LIN {X 0,Y 194.832,Z 950.293,A -85,B 0,C 180,E1 7671.992,E2 7671.992} C_VEL
LIN {X 0,Y 183.693,Z 961.41,A -85,B 0,C 180,E1 7666.758,E2 7666.758} C_VEL
LIN {X 0,Y 173.578,Z 971.355,A -85,B 0,C 180,E1 7660.613,E2 7660.613} C_VEL
LIN {X 0,Y 165.361,Z 979.416,A -85,B 0,C 180,E1 7653.893,E2 7653.893} C_VEL
LIN {X 0,Y 158.738,Z 986.366,A -85,B 0,C 180,E1 7646.018,E2 7646.018} C_VEL
LIN {X 0,Y 154.956,Z 990.985,A -85,B 0,C 180,E1 7638.756,E2 7638.756} C_VEL
LIN {X 0,Y 152.752,Z 994.605,A -85,B 0,C 180,E1 7630.489,E2 7630.489} C_VEL
LIN {X 0,Y 152.139,Z 996.368,A -85,B 0,C 180,E1 7623.866,E2 7623.866} C_VEL
LIN {X 0,Y 152.069,Z 997.179,A -85,B 0,C 180,E1 7618.016,E2 7618.016} C_VEL
LIN {X 0,Y 152.181,Z 997.294,A -85,B 0,C 180,E1 7612.04,E2 7612.04} C_VEL
LIN {X 0,Y 152.864,Z 996.613,A -85,B 0,C 180,E1 7605.477,E2 7605.477} C_VEL
LIN {X 0,Y 155.417,Z 994.355,A -85,B 0,C 180,E1 7596.75,E2 7596.75} C_VEL
LIN {X 0,Y 159.971,Z 990.88,A -85,B 0,C 180,E1 7588.935,E2 7588.935} C_VEL
LIN {X 0,Y 168.381,Z 984.987,A -85,B 0,C 180,E1 7580.226,E2 7580.226} C_VEL
LIN {X 0,Y 178.983,Z 977.818,A -85,B 0,C 180,E1 7572.913,E2 7572.913} C_VEL
LIN {X 0,Y 191.582,Z 968.945,A -85,B 0,C 180,E1 7566.594,E2 7566.594} C_VEL
LIN {X 0,Y 207.009,Z 957.677,A -85,B 0,C 180,E1 7560.794,E2 7560.794} C_VEL
LIN {X 0,Y 222.449,Z 945.698,A -85,B 0,C 180,E1 7556.307,E2 7556.307} C_VEL
LIN {X 0,Y 238.515,Z 932.053,A -85,B 0,C 180,E1 7552.534,E2 7552.534} C_VEL
LIN {X 0,Y 255.431,Z 916.454,A -85,B 0,C 180,E1 7549.29,E2 7549.29} C_VEL
LIN {X 0,Y 271.677,Z 899.924,A -85,B 0,C 180,E1 7546.703,E2 7546.703} C_VEL
LIN {X 0,Y 286.835,Z 882.673,A -85,B 0,C 180,E1 7544.638,E2 7544.638} C_VEL
LIN {X 0,Y 271.407,Z 900.775,A -85,B 0,C 180,E1 7542.66,E2 7542.66} C_VEL
LIN {X 0,Y 266.25,Z 906.214,A -85,B 0,C 180,E1 7542.181,E2 7542.181} C_VEL
LIN {X 0,Y 251.976,Z 920.113,A -85,B 0,C 180,E1 7541.531,E2 7541.531} C_VEL
LIN {X 0,Y 246.66,Z 924.954,A -85,B 0,C 180,E1 7540.925,E2 7540.925} C_VEL
LIN {X 0,Y 229.187,Z 940.666,A -85,B 0,C 180,E1 7537.662,E2 7537.662} C_VEL
LIN {X 0,Y 212.755,Z 954.165,A -85,B 0,C 180,E1 7533.859,E2 7533.859} C_VEL
LIN {X 0,Y 195.426,Z 967.538,A -85,B 0,C 180,E1 7528.708,E2 7528.708} C_VEL
LIN {X 0,Y 181.211,Z 978.023,A -85,B 0,C 180,E1 7523.147,E2 7523.147} C_VEL
LIN {X 0,Y 168.432,Z 987.146,A -85,B 0,C 180,E1 7516.415,E2 7516.415} C_VEL
LIN {X 0,Y 158.156,Z 994.699,A -85,B 0,C 180,E1 7508.757,E2 7508.757} C_VEL
LIN {X 0,Y 150.669,Z 1000.453,A -85,B 0,C 180,E1 7500.298,E2 7500.298} C_VEL
LIN {X 0,Y 146.133,Z 1004.752,A -85,B 0,C 180,E1 7491.272,E2 7491.272} C_VEL
LIN {X 0,Y 144.3,Z 1007.131,A -85,B 0,C 180,E1 7482.821,E2 7482.821} C_VEL
LIN {X 0,Y 144.029,Z 1008.079,A -85,B 0,C 180,E1 7476.387,E2 7476.387} C_VEL
LIN {X 0,Y 144.076,Z 1008.216,A -85,B 0,C 180,E1 7470.408,E2 7470.408} C_VEL
LIN {X 0,Y 144.045,Z 1007.654,A -85,B 0,C 180,E1 7464.833,E2 7464.833} C_VEL
LIN {X 0,Y 144.179,Z 1006.3,A -85,B 0,C 180,E1 7458.814,E2 7458.814} C_VEL
LIN {X 0,Y 145.28,Z 1003.668,A -85,B 0,C 180,E1 7451.555,E2 7451.555} C_VEL
LIN {X 0,Y 148.668,Z 998.874,A -85,B 0,C 180,E1 7442.797,E2 7442.797} C_VEL
LIN {X 0,Y 153.972,Z 992.973,A -85,B 0,C 180,E1 7435.162,E2 7435.162} C_VEL
LIN {X 0,Y 162.295,Z 984.672,A -85,B 0,C 180,E1 7427.352,E2 7427.352} C_VEL
LIN {X 0,Y 172.502,Z 974.948,A -85,B 0,C 180,E1 7420.613,E2 7420.613} C_VEL
LIN {X 0,Y 184.018,Z 963.646,A -85,B 0,C 180,E1 7414.887,E2 7414.887} C_VEL
LIN {X 0,Y 196.383,Z 951.126,A -85,B 0,C 180,E1 7410.075,E2 7410.075} C_VEL
LIN {X 0,Y 208.775,Z 937.625,A -85,B 0,C 180,E1 7406.141,E2 7406.141} C_VEL
LIN {X 0,Y 223.027,Z 920.827,A -85,B 0,C 180,E1 7402.399,E2 7402.399} C_VEL
LIN {X 0,Y 235.885,Z 904.265,A -85,B 0,C 180,E1 7399.563,E2 7399.563} C_VEL
LIN {X 0,Y 248.354,Z 886.236,A -85,B 0,C 180,E1 7397.176,E2 7397.176} C_VEL
LIN {X 0,Y 260.04,Z 867.469,A -85,B 0,C 180,E1 7395.211,E2 7395.211} C_VEL
LIN {X 0,Y 270.544,Z 848.252,A -85,B 0,C 180,E1 7393.628,E2 7393.628} C_VEL
LIN {X 0,Y 280.799,Z 826.787,A -85,B 0,C 180,E1 7392.231,E2 7392.231} C_VEL
LIN {X 0,Y 289.504,Z 805.535,A -85,B 0,C 180,E1 7391.151,E2 7391.151} C_VEL
LIN {X 0,Y 297.135,Z 782.995,A -85,B 0,C 180,E1 7390.273,E2 7390.273} C_VEL
LIN {X 0,Y 303.574,Z 759.689,A -85,B 0,C 180,E1 7389.596,E2 7389.596} C_VEL
LIN {X 0,Y 308.243,Z 736.843,A -85,B 0,C 180,E1 7389.078,E2 7389.078} C_VEL
LIN {X 0,Y 312.449,Z 705.289,A -85,B 0,C 180,E1 7388.469,E2 7388.469} C_VEL
LIN {X 0,Y 324.295,Z 602.682,A -85,B 0,C 180,E1 7386.606,E2 7386.606} C_VEL
LIN {X 0,Y 320.232,Z 595.927,A -85,B 0,C 180,E1 7383.132,E2 7383.132} C_VEL
LIN {X 0,Y 317.949,Z 592.19,A -85,B 0,C 180,E1 7380.805,E2 7380.805} C_VEL
LIN {X 0,Y 315.597,Z 588.414,A -85,B 0,C 180,E1 7378.002,E2 7378.002} C_VEL
LIN {X 0,Y 312.963,Z 584.083,A -85,B 0,C 180,E1 7373.948,E2 7373.948} C_VEL
LIN {X 0,Y 310.602,Z 579.992,A -85,B 0,C 180,E1 7367.23,E2 7367.23} C_VEL
LIN {X 0,Y 310.395,Z 579.187,A -85,B 0,C 180,E1 7365.447,E2 7365.447} C_VEL
LIN {X 0,Y 310.527,Z 579.358,A -85,B 0,C 180,E1 7360.826,E2 7360.826} C_VEL
LIN {X 0,Y 312.556,Z 583.694,A -85,B 0,C 180,E1 7354.007,E2 7354.007} C_VEL
LIN {X 0,Y 313.453,Z 584.799,A -85,B 0,C 180,E1 7352.449,E2 7352.449} C_VEL
LIN {X 0,Y 316.52,Z 589.805,A -85,B 0,C 180,E1 7348.054,E2 7348.054} C_VEL
LIN {X 0,Y 319.481,Z 594.635,A -85,B 0,C 180,E1 7344.84,E2 7344.84} C_VEL
LIN {X 0,Y 323.414,Z 601.079,A -85,B 0,C 180,E1 7341.354,E2 7341.354} C_VEL
LIN {X 0,Y 323.931,Z 602.297,A -85,B 0,C 180,E1 7340.903,E2 7340.903} C_VEL
LIN {X 0,Y 309.802,Z 722.184,A -85,B 0,C 180,E1 7338.744,E2 7338.744} C_VEL
LIN {X 0,Y 305.322,Z 746.033,A -85,B 0,C 180,E1 7338.204,E2 7338.204} C_VEL
LIN {X 0,Y 299.821,Z 768.228,A -85,B 0,C 180,E1 7337.538,E2 7337.538} C_VEL
LIN {X 0,Y 292.969,Z 789.815,A -85,B 0,C 180,E1 7336.686,E2 7336.686} C_VEL
LIN {X 0,Y 284.325,Z 812.53,A -85,B 0,C 180,E1 7335.541,E2 7335.541} C_VEL
LIN {X 0,Y 275.54,Z 832.057,A -85,B 0,C 180,E1 7334.299,E2 7334.299} C_VEL
LIN {X 0,Y 264.822,Z 852.675,A -85,B 0,C 180,E1 7332.656,E2 7332.656} C_VEL
LIN {X 0,Y 253.514,Z 871.813,A -85,B 0,C 180,E1 7330.738,E2 7330.738} C_VEL
LIN {X 0,Y 241.283,Z 889.944,A -85,B 0,C 180,E1 7328.423,E2 7328.423} C_VEL
LIN {X 0,Y 228.308,Z 907.306,A -85,B 0,C 180,E1 7325.614,E2 7325.614} C_VEL
LIN {X 0,Y 215.842,Z 922.349,A -85,B 0,C 180,E1 7322.494,E2 7322.494} C_VEL
LIN {X 0,Y 202.641,Z 936.953,A -85,B 0,C 180,E1 7318.585,E2 7318.585} C_VEL
LIN {X 0,Y 190.981,Z 948.948,A -85,B 0,C 180,E1 7314.421,E2 7314.421} C_VEL
LIN {X 0,Y 178.697,Z 960.792,A -85,B 0,C 180,E1 7308.982,E2 7308.982} C_VEL
LIN {X 0,Y 167.816,Z 971.009,A -85,B 0,C 180,E1 7302.726,E2 7302.726} C_VEL
LIN {X 0,Y 158.765,Z 979.33,A -85,B 0,C 180,E1 7295.698,E2 7295.698} C_VEL
LIN {X 0,Y 151.411,Z 986.537,A -85,B 0,C 180,E1 7287.341,E2 7287.341} C_VEL
LIN {X 0,Y 147.3,Z 991.142,A -85,B 0,C 180,E1 7279.823,E2 7279.823} C_VEL
LIN {X 0,Y 144.836,Z 994.849,A -85,B 0,C 180,E1 7271.047,E2 7271.047} C_VEL
LIN {X 0,Y 144.152,Z 996.634,A -85,B 0,C 180,E1 7264.078,E2 7264.078} C_VEL
LIN {X 0,Y 144.072,Z 997.476,A -85,B 0,C 180,E1 7257.854,E2 7257.854} C_VEL
LIN {X 0,Y 144.21,Z 997.615,A -85,B 0,C 180,E1 7251.581,E2 7251.581} C_VEL
LIN {X 0,Y 144.995,Z 996.975,A -85,B 0,C 180,E1 7244.7,E2 7244.7} C_VEL
LIN {X 0,Y 147.862,Z 994.811,A -85,B 0,C 180,E1 7235.561,E2 7235.561} C_VEL
LIN {X 0,Y 153.044,Z 991.301,A -85,B 0,C 180,E1 7227.216,E2 7227.216} C_VEL
LIN {X 0,Y 162.181,Z 985.516,A -85,B 0,C 180,E1 7218.277,E2 7218.277} C_VEL
LIN {X 0,Y 173.324,Z 978.573,A -85,B 0,C 180,E1 7210.975,E2 7210.975} C_VEL
LIN {X 0,Y 186.679,Z 969.849,A -85,B 0,C 180,E1 7204.609,E2 7204.609} C_VEL
LIN {X 0,Y 201.882,Z 959.492,A -85,B 0,C 180,E1 7199.15,E2 7199.15} C_VEL
LIN {X 0,Y 216.832,Z 948.494,A -85,B 0,C 180,E1 7194.941,E2 7194.941} C_VEL
LIN {X 0,Y 234.646,Z 934.325,A -85,B 0,C 180,E1 7190.93,E2 7190.93} C_VEL
LIN {X 0,Y 251.632,Z 919.547,A -85,B 0,C 180,E1 7187.836,E2 7187.836} C_VEL
LIN {X 0,Y 268.871,Z 902.747,A -85,B 0,C 180,E1 7185.224,E2 7185.224} C_VEL
LIN {X 0,Y 272.667,Z 898.907,A -85,B 0,C 180,E1 7184.682,E2 7184.682} C_VEL
LIN {X 0,Y 256.832,Z 915.179,A -85,B 0,C 180,E1 7182.528,E2 7182.528} C_VEL
LIN {X 0,Y 246.66,Z 924.954,A -85,B 0,C 180,E1 7180.925,E2 7180.925} C_VEL
LIN {X 0,Y 241.229,Z 929.896,A -85,B 0,C 180,E1 7180.269,E2 7180.269} C_VEL
LIN {X 0,Y 225.887,Z 942.079,A -85,B 0,C 180,E1 7179.184,E2 7179.184} C_VEL
LIN {X 0,Y 220.354,Z 946.366,A -85,B 0,C 180,E1 7178.369,E2 7178.369} C_VEL
LIN {X 0,Y 202.342,Z 960.072,A -85,B 0,C 180,E1 7174.084,E2 7174.084} C_VEL
LIN {X 0,Y 185.384,Z 972.199,A -85,B 0,C 180,E1 7168.818,E2 7168.818} C_VEL
LIN {X 0,Y 170.774,Z 981.996,A -85,B 0,C 180,E1 7162.786,E2 7162.786} C_VEL
LIN {X 0,Y 157.16,Z 991.006,A -85,B 0,C 180,E1 7154.937,E2 7154.937} C_VEL
LIN {X 0,Y 147.801,Z 997.325,A -85,B 0,C 180,E1 7147.03,E2 7147.03} C_VEL
LIN {X 0,Y 140.534,Z 1002.714,A -85,B 0,C 180,E1 7137.098,E2 7137.098} C_VEL
LIN {X 0,Y 137.2,Z 1005.822,A -85,B 0,C 180,E1 7128.273,E2 7128.273} C_VEL
LIN {X 0,Y 136.079,Z 1007.586,A -85,B 0,C 180,E1 7119.313,E2 7119.313} C_VEL
LIN {X 0,Y 136.056,Z 1007.968,A -85,B 0,C 180,E1 7112.538,E2 7112.538} C_VEL
LIN {X 0,Y 136.056,Z 1007.622,A -85,B 0,C 180,E1 7106.641,E2 7106.641} C_VEL
LIN {X 0,Y 136.145,Z 1006.248,A -85,B 0,C 180,E1 7099.432,E2 7099.432} C_VEL
LIN {X 0,Y 137.195,Z 1003.721,A -85,B 0,C 180,E1 7091.749,E2 7091.749} C_VEL
LIN {X 0,Y 140.484,Z 999.348,A -85,B 0,C 180,E1 7082.827,E2 7082.827} C_VEL
LIN {X 0,Y 146.158,Z 993.337,A -85,B 0,C 180,E1 7074.459,E2 7074.459} C_VEL
LIN {X 0,Y 154.826,Z 985.253,A -85,B 0,C 180,E1 7066.306,E2 7066.306} C_VEL
LIN {X 0,Y 164.335,Z 976.602,A -85,B 0,C 180,E1 7059.965,E2 7059.965} C_VEL
LIN {X 0,Y 177.145,Z 964.76,A -85,B 0,C 180,E1 7053.581,E2 7053.581} C_VEL
LIN {X 0,Y 190.24,Z 952.141,A -85,B 0,C 180,E1 7048.572,E2 7048.572} C_VEL
LIN {X 0,Y 203.298,Z 938.468,A -85,B 0,C 180,E1 7044.535,E2 7044.535} C_VEL
LIN {X 0,Y 216.778,Z 923.303,A -85,B 0,C 180,E1 7041.085,E2 7041.085} C_VEL
LIN {X 0,Y 229.876,Z 906.972,A -85,B 0,C 180,E1 7038.249,E2 7038.249} C_VEL
LIN {X 0,Y 243.433,Z 888.208,A -85,B 0,C 180,E1 7035.728,E2 7035.728} C_VEL
LIN {X 0,Y 255.742,Z 869.143,A -85,B 0,C 180,E1 7033.734,E2 7033.734} C_VEL
LIN {X 0,Y 267.046,Z 849.002,A -85,B 0,C 180,E1 7032.102,E2 7032.102} C_VEL
LIN {X 0,Y 277.766,Z 827.118,A -85,B 0,C 180,E1 7030.713,E2 7030.713} C_VEL
LIN {X 0,Y 286.504,Z 806.21,A -85,B 0,C 180,E1 7029.681,E2 7029.681} C_VEL
LIN {X 0,Y 294.402,Z 783.436,A -85,B 0,C 180,E1 7028.819,E2 7028.819} C_VEL
LIN {X 0,Y 300.942,Z 760.311,A -85,B 0,C 180,E1 7028.167,E2 7028.167} C_VEL
LIN {X 0,Y 305.784,Z 737.07,A -85,B 0,C 180,E1 7027.657,E2 7027.657} C_VEL
LIN {X 0,Y 310.085,Z 705.601,A -85,B 0,C 180,E1 7027.063,E2 7027.063} C_VEL
LIN {X 0,Y 321.529,Z 608.329,A -85,B 0,C 180,E1 7025.352,E2 7025.352} C_VEL
LIN {X 0,Y 317.312,Z 601.015,A -85,B 0,C 180,E1 7021.354,E2 7021.354} C_VEL
LIN {X 0,Y 314.291,Z 596.237,A -85,B 0,C 180,E1 7017.812,E2 7017.812} C_VEL
LIN {X 0,Y 311.709,Z 591.924,A -85,B 0,C 180,E1 7013.738,E2 7013.738} C_VEL
LIN {X 0,Y 309.455,Z 587.902,A -85,B 0,C 180,E1 7007.118,E2 7007.118} C_VEL
LIN {X 0,Y 309.262,Z 587.103,A -85,B 0,C 180,E1 7005.393,E2 7005.393} C_VEL
LIN {X 0,Y 309.401,Z 587.346,A -85,B 0,C 180,E1 7000.754,E2 7000.754} C_VEL
LIN {X 0,Y 311.174,Z 591.374,A -85,B 0,C 180,E1 6994.496,E2 6994.496} C_VEL
LIN {X 0,Y 312.197,Z 592.659,A -85,B 0,C 180,E1 6992.639,E2 6992.639} C_VEL
LIN {X 0,Y 315.136,Z 597.553,A -85,B 0,C 180,E1 6988.325,E2 6988.325} C_VEL
LIN {X 0,Y 318.002,Z 602.339,A -85,B 0,C 180,E1 6985.137,E2 6985.137} C_VEL
LIN {X 0,Y 321.19,Z 607.752,A -85,B 0,C 180,E1 6982.187,E2 6982.187} C_VEL
LIN {X 0,Y 307.433,Z 722.444,A -85,B 0,C 180,E1 6980.162,E2 6980.162} C_VEL
LIN {X 0,Y 302.898,Z 746.237,A -85,B 0,C 180,E1 6979.641,E2 6979.641} C_VEL
LIN {X 0,Y 297.363,Z 768.273,A -85,B 0,C 180,E1 6979.003,E2 6979.003} C_VEL
LIN {X 0,Y 290.411,Z 789.843,A -85,B 0,C 180,E1 6978.182,E2 6978.182} C_VEL
LIN {X 0,Y 281.81,Z 812.156,A -85,B 0,C 180,E1 6977.1,E2 6977.1} C_VEL
LIN {X 0,Y 272.857,Z 831.753,A -85,B 0,C 180,E1 6975.898,E2 6975.898} C_VEL
LIN {X 0,Y 261.699,Z 852.86,A -85,B 0,C 180,E1 6974.27,E2 6974.27} C_VEL
LIN {X 0,Y 249.952,Z 872.361,A -85,B 0,C 180,E1 6972.369,E2 6972.369} C_VEL
LIN {X 0,Y 237.434,Z 890.496,A -85,B 0,C 180,E1 6970.103,E2 6970.103} C_VEL
LIN {X 0,Y 224.118,Z 907.857,A -85,B 0,C 180,E1 6967.344,E2 6967.344} C_VEL
LIN {X 0,Y 211.285,Z 922.885,A -85,B 0,C 180,E1 6964.263,E2 6964.263} C_VEL
LIN {X 0,Y 197.639,Z 937.451,A -85,B 0,C 180,E1 6960.381,E2 6960.381} C_VEL
LIN {X 0,Y 184.89,Z 950.09,A -85,B 0,C 180,E1 6955.969,E2 6955.969} C_VEL
LIN {X 0,Y 172.619,Z 961.369,A -85,B 0,C 180,E1 6950.681,E2 6950.681} C_VEL
LIN {X 0,Y 161.281,Z 971.477,A -85,B 0,C 180,E1 6944.348,E2 6944.348} C_VEL
LIN {X 0,Y 151.792,Z 979.707,A -85,B 0,C 180,E1 6937.179,E2 6937.179} C_VEL
LIN {X 0,Y 143.882,Z 986.946,A -85,B 0,C 180,E1 6928.397,E2 6928.397} C_VEL
LIN {X 0,Y 139.484,Z 991.535,A -85,B 0,C 180,E1 6920.5,E2 6920.5} C_VEL
LIN {X 0,Y 136.856,Z 995.203,A -85,B 0,C 180,E1 6911.238,E2 6911.238} C_VEL
LIN {X 0,Y 136.147,Z 996.973,A -85,B 0,C 180,E1 6903.844,E2 6903.844} C_VEL
LIN {X 0,Y 136.075,Z 997.777,A -85,B 0,C 180,E1 6897.55,E2 6897.55} C_VEL
LIN {X 0,Y 136.243,Z 997.939,A -85,B 0,C 180,E1 6891.072,E2 6891.072} C_VEL
LIN {X 0,Y 137.162,Z 997.335,A -85,B 0,C 180,E1 6883.794,E2 6883.794} C_VEL
LIN {X 0,Y 140.373,Z 995.277,A -85,B 0,C 180,E1 6874.245,E2 6874.245} C_VEL
LIN {X 0,Y 146.175,Z 991.795,A -85,B 0,C 180,E1 6865.438,E2 6865.438} C_VEL
LIN {X 0,Y 156.187,Z 986.085,A -85,B 0,C 180,E1 6856.181,E2 6856.181} C_VEL
LIN {X 0,Y 168.818,Z 978.845,A -85,B 0,C 180,E1 6848.424,E2 6848.424} C_VEL
LIN {X 0,Y 183.116,Z 970.124,A -85,B 0,C 180,E1 6842.097,E2 6842.097} C_VEL
LIN {X 0,Y 199.318,Z 959.7,A -85,B 0,C 180,E1 6836.715,E2 6836.715} C_VEL
LIN {X 0,Y 215.447,Z 948.401,A -85,B 0,C 180,E1 6832.535,E2 6832.535} C_VEL
LIN {X 0,Y 233.421,Z 934.669,A -85,B 0,C 180,E1 6828.812,E2 6828.812} C_VEL
LIN {X 0,Y 250.67,Z 920.224,A -85,B 0,C 180,E1 6825.919,E2 6825.919} C_VEL
LIN {X 0,Y 258.508,Z 913.046,A -85,B 0,C 180,E1 6824.752,E2 6824.752} C_VEL
LIN {X 0,Y 241.477,Z 928.765,A -85,B 0,C 180,E1 6822.252,E2 6822.252} C_VEL
LIN {X 0,Y 223.758,Z 943.608,A -85,B 0,C 180,E1 6819.066,E2 6819.066} C_VEL
LIN {X 0,Y 220.354,Z 946.366,A -85,B 0,C 180,E1 6818.369,E2 6818.369} C_VEL
LIN {X 0,Y 214.771,Z 950.617,A -85,B 0,C 180,E1 6817.487,E2 6817.487} C_VEL
LIN {X 0,Y 198.781,Z 961.182,A -85,B 0,C 180,E1 6815.791,E2 6815.791} C_VEL
LIN {X 0,Y 193.104,Z 964.791,A -85,B 0,C 180,E1 6814.666,E2 6814.666} C_VEL
LIN {X 0,Y 176.188,Z 975.809,A -85,B 0,C 180,E1 6809.288,E2 6809.288} C_VEL
LIN {X 0,Y 159.726,Z 986.02,A -85,B 0,C 180,E1 6802.081,E2 6802.081} C_VEL
LIN {X 0,Y 146.511,Z 994.111,A -85,B 0,C 180,E1 6793.666,E2 6793.666} C_VEL
LIN {X 0,Y 136.907,Z 1000.051,A -85,B 0,C 180,E1 6784.23,E2 6784.23} C_VEL
LIN {X 0,Y 130.704,Z 1004.496,A -85,B 0,C 180,E1 6773.371,E2 6773.371} C_VEL
LIN {X 0,Y 128.478,Z 1006.637,A -85,B 0,C 180,E1 6764.432,E2 6764.432} C_VEL
LIN {X 0,Y 128.037,Z 1007.576,A -85,B 0,C 180,E1 6756.288,E2 6756.288} C_VEL
LIN {X 0,Y 128.09,Z 1007.539,A -85,B 0,C 180,E1 6749.565,E2 6749.565} C_VEL
LIN {X 0,Y 128.05,Z 1006.691,A -85,B 0,C 180,E1 6742.582,E2 6742.582} C_VEL
LIN {X 0,Y 128.77,Z 1004.438,A -85,B 0,C 180,E1 6733.781,E2 6733.781} C_VEL
LIN {X 0,Y 131.207,Z 1000.907,A -85,B 0,C 180,E1 6725.234,E2 6725.234} C_VEL
LIN {X 0,Y 136.395,Z 995.606,A -85,B 0,C 180,E1 6716.157,E2 6716.157} C_VEL
LIN {X 0,Y 144.237,Z 988.47,A -85,B 0,C 180,E1 6707.763,E2 6707.763} C_VEL
LIN {X 0,Y 154.54,Z 979.684,A -85,B 0,C 180,E1 6700.248,E2 6700.248} C_VEL
LIN {X 0,Y 165.702,Z 969.975,A -85,B 0,C 180,E1 6694.261,E2 6694.261} C_VEL
LIN {X 0,Y 179.743,Z 957.256,A -85,B 0,C 180,E1 6688.511,E2 6688.511} C_VEL
LIN {X 0,Y 192.967,Z 944.44,A -85,B 0,C 180,E1 6684.248,E2 6684.248} C_VEL
LIN {X 0,Y 207.087,Z 929.495,A -85,B 0,C 180,E1 6680.527,E2 6680.527} C_VEL
LIN {X 0,Y 220.687,Z 913.83,A -85,B 0,C 180,E1 6677.532,E2 6677.532} C_VEL
LIN {X 0,Y 233.937,Z 896.685,A -85,B 0,C 180,E1 6675.03,E2 6675.03} C_VEL
LIN {X 0,Y 247.299,Z 877.408,A -85,B 0,C 180,E1 6672.848,E2 6672.848} C_VEL
LIN {X 0,Y 258.846,Z 858.522,A -85,B 0,C 180,E1 6671.186,E2 6671.186} C_VEL
LIN {X 0,Y 269.837,Z 837.889,A -85,B 0,C 180,E1 6669.766,E2 6669.766} C_VEL
LIN {X 0,Y 279.521,Z 817.029,A -85,B 0,C 180,E1 6668.64,E2 6668.64} C_VEL
LIN {X 0,Y 288.038,Z 794.958,A -85,B 0,C 180,E1 6667.727,E2 6667.727} C_VEL
LIN {X 0,Y 295.615,Z 771.189,A -85,B 0,C 180,E1 6666.985,E2 6666.985} C_VEL
LIN {X 0,Y 301.259,Z 748.585,A -85,B 0,C 180,E1 6666.451,E2 6666.451} C_VEL
LIN {X 0,Y 305.459,Z 724.638,A -85,B 0,C 180,E1 6665.976,E2 6665.976} C_VEL
LIN {X 0,Y 318.866,Z 614.103,A -85,B 0,C 180,E1 6664.045,E2 6664.045} C_VEL
LIN {X 0,Y 315.202,Z 607.785,A -85,B 0,C 180,E1 6660.363,E2 6660.363} C_VEL
LIN {X 0,Y 312.845,Z 603.886,A -85,B 0,C 180,E1 6657.435,E2 6657.435} C_VEL
LIN {X 0,Y 310.459,Z 599.764,A -85,B 0,C 180,E1 6653.527,E2 6653.527} C_VEL
LIN {X 0,Y 308.303,Z 595.714,A -85,B 0,C 180,E1 6646.878,E2 6646.878} C_VEL
LIN {X 0,Y 308.101,Z 594.982,A -85,B 0,C 180,E1 6644.952,E2 6644.952} C_VEL
LIN {X 0,Y 308.26,Z 595.245,A -85,B 0,C 180,E1 6640.876,E2 6640.876} C_VEL
LIN {X 0,Y 310.088,Z 599.376,A -85,B 0,C 180,E1 6634.4,E2 6634.4} C_VEL
LIN {X 0,Y 310.937,Z 600.517,A -85,B 0,C 180,E1 6632.83,E2 6632.83} C_VEL
LIN {X 0,Y 313.751,Z 605.286,A -85,B 0,C 180,E1 6628.608,E2 6628.608} C_VEL
LIN {X 0,Y 316.502,Z 609.991,A -85,B 0,C 180,E1 6625.465,E2 6625.465} C_VEL
LIN {X 0,Y 318.537,Z 613.657,A -85,B 0,C 180,E1 6623.475,E2 6623.475} C_VEL
LIN {X 0,Y 305.142,Z 722.86,A -85,B 0,C 180,E1 6621.594,E2 6621.594} C_VEL
LIN {X 0,Y 300.517,Z 746.67,A -85,B 0,C 180,E1 6621.089,E2 6621.089} C_VEL
LIN {X 0,Y 294.648,Z 769.471,A -85,B 0,C 180,E1 6620.447,E2 6620.447} C_VEL
LIN {X 0,Y 287.809,Z 790.341,A -85,B 0,C 180,E1 6619.679,E2 6619.679} C_VEL
LIN {X 0,Y 278.977,Z 812.85,A -85,B 0,C 180,E1 6618.622,E2 6618.622} C_VEL
LIN {X 0,Y 269.6,Z 833.002,A -85,B 0,C 180,E1 6617.422,E2 6617.422} C_VEL
LIN {X 0,Y 258.585,Z 853.385,A -85,B 0,C 180,E1 6615.892,E2 6615.892} C_VEL
LIN {X 0,Y 247.01,Z 872.22,A -85,B 0,C 180,E1 6614.115,E2 6614.115} C_VEL
LIN {X 0,Y 234.195,Z 890.427,A -85,B 0,C 180,E1 6611.914,E2 6611.914} C_VEL
LIN {X 0,Y 220.922,Z 907.387,A -85,B 0,C 180,E1 6609.307,E2 6609.307} C_VEL
LIN {X 0,Y 207.693,Z 922.516,A -85,B 0,C 180,E1 6606.298,E2 6606.298} C_VEL
LIN {X 0,Y 192.838,Z 937.934,A -85,B 0,C 180,E1 6602.269,E2 6602.269} C_VEL
LIN {X 0,Y 179.608,Z 950.579,A -85,B 0,C 180,E1 6597.869,E2 6597.869} C_VEL
LIN {X 0,Y 166.632,Z 961.969,A -85,B 0,C 180,E1 6592.47,E2 6592.47} C_VEL
LIN {X 0,Y 154.882,Z 971.905,A -85,B 0,C 180,E1 6586.106,E2 6586.106} C_VEL
LIN {X 0,Y 145.269,Z 979.771,A -85,B 0,C 180,E1 6579.098,E2 6579.098} C_VEL
LIN {X 0,Y 136.986,Z 986.856,A -85,B 0,C 180,E1 6570.351,E2 6570.351} C_VEL
LIN {X 0,Y 132.084,Z 991.489,A -85,B 0,C 180,E1 6562.157,E2 6562.157} C_VEL
LIN {X 0,Y 129.135,Z 995.182,A -85,B 0,C 180,E1 6552.877,E2 6552.877} C_VEL
LIN {X 0,Y 128.182,Z 997.15,A -85,B 0,C 180,E1 6544.583,E2 6544.583} C_VEL
LIN {X 0,Y 128.082,Z 998.031,A -85,B 0,C 180,E1 6537.926,E2 6537.926} C_VEL
LIN {X 0,Y 128.263,Z 998.272,A -85,B 0,C 180,E1 6530.831,E2 6530.831} C_VEL
LIN {X 0,Y 129.358,Z 997.697,A -85,B 0,C 180,E1 6522.738,E2 6522.738} C_VEL
LIN {X 0,Y 133.033,Z 995.719,A -85,B 0,C 180,E1 6512.654,E2 6512.654} C_VEL
LIN {X 0,Y 139.735,Z 992.164,A -85,B 0,C 180,E1 6503.177,E2 6503.177} C_VEL
LIN {X 0,Y 150.542,Z 986.611,A -85,B 0,C 180,E1 6493.835,E2 6493.835} C_VEL
LIN {X 0,Y 163.467,Z 979.772,A -85,B 0,C 180,E1 6486.322,E2 6486.322} C_VEL
LIN {X 0,Y 179.404,Z 970.759,A -85,B 0,C 180,E1 6479.682,E2 6479.682} C_VEL
LIN {X 0,Y 196.974,Z 960.091,A -85,B 0,C 180,E1 6474.274,E2 6474.274} C_VEL
LIN {X 0,Y 214.125,Z 948.636,A -85,B 0,C 180,E1 6470.181,E2 6470.181} C_VEL
LIN {X 0,Y 233.026,Z 934.733,A -85,B 0,C 180,E1 6466.604,E2 6466.604} C_VEL
LIN {X 0,Y 244.255,Z 925.776,A -85,B 0,C 180,E1 6464.813,E2 6464.813} C_VEL
LIN {X 0,Y 224.406,Z 942.034,A -85,B 0,C 180,E1 6461.644,E2 6461.644} C_VEL
LIN {X 0,Y 207.267,Z 954.887,A -85,B 0,C 180,E1 6458.196,E2 6458.196} C_VEL
LIN {X 0,Y 193.104,Z 964.791,A -85,B 0,C 180,E1 6454.666,E2 6454.666} C_VEL
LIN {X 0,Y 187.429,Z 968.291,A -85,B 0,C 180,E1 6453.451,E2 6453.451} C_VEL
LIN {X 0,Y 170.37,Z 977.521,A -85,B 0,C 180,E1 6450.674,E2 6450.674} C_VEL
LIN {X 0,Y 165.715,Z 979.973,A -85,B 0,C 180,E1 6449.308,E2 6449.308} C_VEL
LIN {X 0,Y 150.461,Z 988.695,A -85,B 0,C 180,E1 6442.273,E2 6442.273} C_VEL
LIN {X 0,Y 137.593,Z 995.744,A -85,B 0,C 180,E1 6433.67,E2 6433.67} C_VEL
LIN {X 0,Y 128.081,Z 1001.229,A -85,B 0,C 180,E1 6423.672,E2 6423.672} C_VEL
LIN {X 0,Y 122.662,Z 1004.667,A -85,B 0,C 180,E1 6413.554,E2 6413.554} C_VEL
LIN {X 0,Y 120.346,Z 1006.724,A -85,B 0,C 180,E1 6403.464,E2 6403.464} C_VEL
LIN {X 0,Y 120.041,Z 1007.369,A -85,B 0,C 180,E1 6394.79,E2 6394.79} C_VEL
LIN {X 0,Y 120.089,Z 1007.146,A -85,B 0,C 180,E1 6388.104,E2 6388.104} C_VEL
LIN {X 0,Y 120.116,Z 1006.004,A -85,B 0,C 180,E1 6380.43,E2 6380.43} C_VEL
LIN {X 0,Y 121.23,Z 1003.467,A -85,B 0,C 180,E1 6371.251,E2 6371.251} C_VEL
LIN {X 0,Y 124.492,Z 999.65,A -85,B 0,C 180,E1 6362.06,E2 6362.06} C_VEL
LIN {X 0,Y 130.97,Z 993.695,A -85,B 0,C 180,E1 6352.373,E2 6352.373} C_VEL
LIN {X 0,Y 139.572,Z 986.653,A -85,B 0,C 180,E1 6344.262,E2 6344.262} C_VEL
LIN {X 0,Y 150.988,Z 977.388,A -85,B 0,C 180,E1 6336.768,E2 6336.768} C_VEL
LIN {X 0,Y 163.777,Z 966.846,A -85,B 0,C 180,E1 6330.614,E2 6330.614} C_VEL
LIN {X 0,Y 177.34,Z 954.816,A -85,B 0,C 180,E1 6325.589,E2 6325.589} C_VEL
LIN {X 0,Y 192.026,Z 940.864,A -85,B 0,C 180,E1 6321.273,E2 6321.273} C_VEL
LIN {X 0,Y 205.098,Z 927.225,A -85,B 0,C 180,E1 6318.108,E2 6318.108} C_VEL
LIN {X 0,Y 219.802,Z 910.313,A -85,B 0,C 180,E1 6315.115,E2 6315.115} C_VEL
LIN {X 0,Y 233.22,Z 893.131,A -85,B 0,C 180,E1 6312.79,E2 6312.79} C_VEL
LIN {X 0,Y 246.01,Z 874.576,A -85,B 0,C 180,E1 6310.855,E2 6310.855} C_VEL
LIN {X 0,Y 258.267,Z 854.548,A -85,B 0,C 180,E1 6309.223,E2 6309.223} C_VEL
LIN {X 0,Y 269.005,Z 834.209,A -85,B 0,C 180,E1 6307.938,E2 6307.938} C_VEL
LIN {X 0,Y 278.925,Z 812.354,A -85,B 0,C 180,E1 6306.866,E2 6306.866} C_VEL
LIN {X 0,Y 287.21,Z 790.727,A -85,B 0,C 180,E1 6306.047,E2 6306.047} C_VEL
LIN {X 0,Y 294.353,Z 767.598,A -85,B 0,C 180,E1 6305.399,E2 6305.399} C_VEL
LIN {X 0,Y 300.074,Z 743.844,A -85,B 0,C 180,E1 6304.883,E2 6304.883} C_VEL
LIN {X 0,Y 303.899,Z 720.855,A -85,B 0,C 180,E1 6304.452,E2 6304.452} C_VEL
LIN {X 0,Y 316.262,Z 619.78,A -85,B 0,C 180,E1 6302.718,E2 6302.718} C_VEL
LIN {X 0,Y 313.47,Z 615.029,A -85,B 0,C 180,E1 6299.725,E2 6299.725} C_VEL
LIN {X 0,Y 311.55,Z 611.71,A -85,B 0,C 180,E1 6297.24,E2 6297.24} C_VEL
LIN {X 0,Y 309.213,Z 607.604,A -85,B 0,C 180,E1 6293.315,E2 6293.315} C_VEL
LIN {X 0,Y 307.137,Z 603.523,A -85,B 0,C 180,E1 6286.636,E2 6286.636} C_VEL
LIN {X 0,Y 306.959,Z 602.876,A -85,B 0,C 180,E1 6284.589,E2 6284.589} C_VEL
LIN {X 0,Y 307.121,Z 603.146,A -85,B 0,C 180,E1 6281,E2 6281} C_VEL
LIN {X 0,Y 308.906,Z 607.271,A -85,B 0,C 180,E1 6274.501,E2 6274.501} C_VEL
LIN {X 0,Y 309.629,Z 608.251,A -85,B 0,C 180,E1 6273.122,E2 6273.122} C_VEL
LIN {X 0,Y 312.389,Z 613.047,A -85,B 0,C 180,E1 6268.874,E2 6268.874} C_VEL
LIN {X 0,Y 315.085,Z 617.779,A -85,B 0,C 180,E1 6265.718,E2 6265.718} C_VEL
LIN {X 0,Y 315.985,Z 619.42,A -85,B 0,C 180,E1 6264.787,E2 6264.787} C_VEL
LIN {X 0,Y 303.023,Z 723.317,A -85,B 0,C 180,E1 6263.045,E2 6263.045} C_VEL
LIN {X 0,Y 298.33,Z 747.077,A -85,B 0,C 180,E1 6262.559,E2 6262.559} C_VEL
LIN {X 0,Y 292.57,Z 769.227,A -85,B 0,C 180,E1 6261.963,E2 6261.963} C_VEL
LIN {X 0,Y 285.404,Z 790.779,A -85,B 0,C 180,E1 6261.203,E2 6261.203} C_VEL
LIN {X 0,Y 276.077,Z 814.035,A -85,B 0,C 180,E1 6260.145,E2 6260.145} C_VEL
LIN {X 0,Y 266.385,Z 834.424,A -85,B 0,C 180,E1 6258.966,E2 6258.966} C_VEL
LIN {X 0,Y 255.042,Z 854.825,A -85,B 0,C 180,E1 6257.468,E2 6257.468} C_VEL
LIN {X 0,Y 243.02,Z 873.875,A -85,B 0,C 180,E1 6255.705,E2 6255.705} C_VEL
LIN {X 0,Y 230.36,Z 891.41,A -85,B 0,C 180,E1 6253.629,E2 6253.629} C_VEL
LIN {X 0,Y 215.555,Z 909.688,A -85,B 0,C 180,E1 6250.835,E2 6250.835} C_VEL
LIN {X 0,Y 202.019,Z 924.66,A -85,B 0,C 180,E1 6247.848,E2 6247.848} C_VEL
LIN {X 0,Y 187.507,Z 939.067,A -85,B 0,C 180,E1 6244.038,E2 6244.038} C_VEL
LIN {X 0,Y 173.499,Z 951.896,A -85,B 0,C 180,E1 6239.516,E2 6239.516} C_VEL
LIN {X 0,Y 160.532,Z 962.776,A -85,B 0,C 180,E1 6234.261,E2 6234.261} C_VEL
LIN {X 0,Y 147.54,Z 973.153,A -85,B 0,C 180,E1 6227.337,E2 6227.337} C_VEL
LIN {X 0,Y 137.552,Z 980.914,A -85,B 0,C 180,E1 6220.035,E2 6220.035} C_VEL
LIN {X 0,Y 128.993,Z 987.734,A -85,B 0,C 180,E1 6210.877,E2 6210.877} C_VEL
LIN {X 0,Y 123.919,Z 992.298,A -85,B 0,C 180,E1 6202.104,E2 6202.104} C_VEL
LIN {X 0,Y 120.898,Z 995.9,A -85,B 0,C 180,E1 6191.671,E2 6191.671} C_VEL
LIN {X 0,Y 120.154,Z 997.562,A -85,B 0,C 180,E1 6183.817,E2 6183.817} C_VEL
LIN {X 0,Y 120.085,Z 998.353,A -85,B 0,C 180,E1 6177.221,E2 6177.221} C_VEL
LIN {X 0,Y 120.366,Z 998.584,A -85,B 0,C 180,E1 6169.6,E2 6169.6} C_VEL
LIN {X 0,Y 121.761,Z 997.995,A -85,B 0,C 180,E1 6160.917,E2 6160.917} C_VEL
LIN {X 0,Y 126.372,Z 995.872,A -85,B 0,C 180,E1 6149.9,E2 6149.9} C_VEL
LIN {X 0,Y 134.18,Z 992.263,A -85,B 0,C 180,E1 6140.047,E2 6140.047} C_VEL
LIN {X 0,Y 146.448,Z 986.535,A -85,B 0,C 180,E1 6130.489,E2 6130.489} C_VEL
LIN {X 0,Y 161.192,Z 979.367,A -85,B 0,C 180,E1 6122.814,E2 6122.814} C_VEL
LIN {X 0,Y 178.341,Z 970.179,A -85,B 0,C 180,E1 6116.43,E2 6116.43} C_VEL
LIN {X 0,Y 197.304,Z 959.111,A -85,B 0,C 180,E1 6111.22,E2 6111.22} C_VEL
LIN {X 0,Y 216.49,Z 946.788,A -85,B 0,C 180,E1 6107.193,E2 6107.193} C_VEL
LIN {X 0,Y 229.959,Z 937.223,A -85,B 0,C 180,E1 6104.869,E2 6104.869} C_VEL
LIN {X 0,Y 210.766,Z 951.299,A -85,B 0,C 180,E1 6101.6,E2 6101.6} C_VEL
LIN {X 0,Y 192.511,Z 963.682,A -85,B 0,C 180,E1 6097.608,E2 6097.608} C_VEL
LIN {X 0,Y 173.959,Z 975.125,A -85,B 0,C 180,E1 6092.283,E2 6092.283} C_VEL
LIN {X 0,Y 165.715,Z 979.973,A -85,B 0,C 180,E1 6089.308,E2 6089.308} C_VEL
LIN {X 0,Y 160.272,Z 982.892,A -85,B 0,C 180,E1 6087.626,E2 6087.626} C_VEL
LIN {X 0,Y 144.489,Z 989.665,A -85,B 0,C 180,E1 6083.682,E2 6083.682} C_VEL
LIN {X 0,Y 139.45,Z 991.898,A -85,B 0,C 180,E1 6081.492,E2 6081.492} C_VEL
LIN {X 0,Y 126.436,Z 998.42,A -85,B 0,C 180,E1 6071.641,E2 6071.641} C_VEL
LIN {X 0,Y 118.144,Z 1002.784,A -85,B 0,C 180,E1 6061.269,E2 6061.269} C_VEL
LIN {X 0,Y 113.372,Z 1005.668,A -85,B 0,C 180,E1 6049.594,E2 6049.594} C_VEL
LIN {X 0,Y 112.114,Z 1006.8,A -85,B 0,C 180,E1 6040.288,E2 6040.288} C_VEL
LIN {X 0,Y 112.064,Z 1006.99,A -85,B 0,C 180,E1 6033.082,E2 6033.082} C_VEL
LIN {X 0,Y 112.078,Z 1006.646,A -85,B 0,C 180,E1 6026.945,E2 6026.945} C_VEL
LIN {X 0,Y 112.162,Z 1005.466,A -85,B 0,C 180,E1 6019.224,E2 6019.224} C_VEL
LIN {X 0,Y 113.497,Z 1002.992,A -85,B 0,C 180,E1 6009.92,E2 6009.92} C_VEL
LIN {X 0,Y 117.66,Z 998.749,A -85,B 0,C 180,E1 5999.361,E2 5999.361} C_VEL
LIN {X 0,Y 124.947,Z 992.644,A -85,B 0,C 180,E1 5989.481,E2 5989.481} C_VEL
LIN {X 0,Y 134.903,Z 985.106,A -85,B 0,C 180,E1 5980.907,E2 5980.907} C_VEL
LIN {X 0,Y 146.727,Z 976.035,A -85,B 0,C 180,E1 5973.783,E2 5973.783} C_VEL
LIN {X 0,Y 161.068,Z 964.611,A -85,B 0,C 180,E1 5967.439,E2 5967.439} C_VEL
LIN {X 0,Y 174.627,Z 953.017,A -85,B 0,C 180,E1 5962.831,E2 5962.831} C_VEL
LIN {X 0,Y 189.934,Z 938.705,A -85,B 0,C 180,E1 5958.668,E2 5958.668} C_VEL
LIN {X 0,Y 204.826,Z 923.455,A -85,B 0,C 180,E1 5955.374,E2 5955.374} C_VEL
LIN {X 0,Y 219.296,Z 906.76,A -85,B 0,C 180,E1 5952.694,E2 5952.694} C_VEL
LIN {X 0,Y 233.779,Z 888.076,A -85,B 0,C 180,E1 5950.408,E2 5950.408} C_VEL
LIN {X 0,Y 246.258,Z 869.853,A -85,B 0,C 180,E1 5948.691,E2 5948.691} C_VEL
LIN {X 0,Y 257.994,Z 850.247,A -85,B 0,C 180,E1 5947.255,E2 5947.255} C_VEL
LIN {X 0,Y 268.449,Z 830.388,A -85,B 0,C 180,E1 5946.105,E2 5946.105} C_VEL
LIN {X 0,Y 278.044,Z 808.781,A -85,B 0,C 180,E1 5945.143,E2 5945.143} C_VEL
LIN {X 0,Y 286.747,Z 785.439,A -85,B 0,C 180,E1 5944.346,E2 5944.346} C_VEL
LIN {X 0,Y 293.469,Z 763.136,A -85,B 0,C 180,E1 5943.787,E2 5943.787} C_VEL
LIN {X 0,Y 298.89,Z 739.343,A -85,B 0,C 180,E1 5943.316,E2 5943.316} C_VEL
LIN {X 0,Y 302.755,Z 714.889,A -85,B 0,C 180,E1 5942.88,E2 5942.88} C_VEL
LIN {X 0,Y 313.824,Z 625.838,A -85,B 0,C 180,E1 5941.414,E2 5941.414} C_VEL
LIN {X 0,Y 311.636,Z 622.004,A -85,B 0,C 180,E1 5938.896,E2 5938.896} C_VEL
LIN {X 0,Y 310.124,Z 619.357,A -85,B 0,C 180,E1 5936.858,E2 5936.858} C_VEL
LIN {X 0,Y 307.972,Z 615.442,A -85,B 0,C 180,E1 5933.1,E2 5933.1} C_VEL
LIN {X 0,Y 305.973,Z 611.331,A -85,B 0,C 180,E1 5926.391,E2 5926.391} C_VEL
LIN {X 0,Y 305.825,Z 610.794,A -85,B 0,C 180,E1 5924.254,E2 5924.254} C_VEL
LIN {X 0,Y 305.985,Z 611.196,A -85,B 0,C 180,E1 5920.927,E2 5920.927} C_VEL
LIN {X 0,Y 307.821,Z 615.271,A -85,B 0,C 180,E1 5914.404,E2 5914.404} C_VEL
LIN {X 0,Y 308.475,Z 616.352,A -85,B 0,C 180,E1 5913.117,E2 5913.117} C_VEL
LIN {X 0,Y 311.058,Z 620.861,A -85,B 0,C 180,E1 5909.107,E2 5909.107} C_VEL
LIN {X 0,Y 313.542,Z 625.311,A -85,B 0,C 180,E1 5906.121,E2 5906.121} C_VEL
LIN {X 0,Y 301.031,Z 723.601,A -85,B 0,C 180,E1 5904.514,E2 5904.514} C_VEL
LIN {X 0,Y 296.273,Z 747.339,A -85,B 0,C 180,E1 5904.049,E2 5904.049} C_VEL
LIN {X 0,Y 290.233,Z 770.126,A -85,B 0,C 180,E1 5903.459,E2 5903.459} C_VEL
LIN {X 0,Y 282.998,Z 791.554,A -85,B 0,C 180,E1 5902.733,E2 5902.733} C_VEL
LIN {X 0,Y 273.726,Z 814.321,A -85,B 0,C 180,E1 5901.741,E2 5901.741} C_VEL
LIN {X 0,Y 263.575,Z 835.36,A -85,B 0,C 180,E1 5900.573,E2 5900.573} C_VEL
LIN {X 0,Y 252.34,Z 855.189,A -85,B 0,C 180,E1 5899.172,E2 5899.172} C_VEL
LIN {X 0,Y 240.086,Z 874.24,A -85,B 0,C 180,E1 5897.476,E2 5897.476} C_VEL
LIN {X 0,Y 227.158,Z 891.775,A -85,B 0,C 180,E1 5895.473,E2 5895.473} C_VEL
LIN {X 0,Y 211.998,Z 910.045,A -85,B 0,C 180,E1 5892.766,E2 5892.766} C_VEL
LIN {X 0,Y 197.758,Z 925.4,A -85,B 0,C 180,E1 5889.779,E2 5889.779} C_VEL
LIN {X 0,Y 183.13,Z 939.467,A -85,B 0,C 180,E1 5886.121,E2 5886.121} C_VEL
LIN {X 0,Y 168.953,Z 952.024,A -85,B 0,C 180,E1 5881.771,E2 5881.771} C_VEL
LIN {X 0,Y 155.078,Z 963.18,A -85,B 0,C 180,E1 5876.404,E2 5876.404} C_VEL
LIN {X 0,Y 141.413,Z 973.535,A -85,B 0,C 180,E1 5869.397,E2 5869.397} C_VEL
LIN {X 0,Y 130.78,Z 981.324,A -85,B 0,C 180,E1 5861.867,E2 5861.867} C_VEL
LIN {X 0,Y 121.651,Z 988.103,A -85,B 0,C 180,E1 5852.343,E2 5852.343} C_VEL
LIN {X 0,Y 115.96,Z 992.881,A -85,B 0,C 180,E1 5842.556,E2 5842.556} C_VEL
LIN {X 0,Y 112.922,Z 996.239,A -85,B 0,C 180,E1 5831.933,E2 5831.933} C_VEL
LIN {X 0,Y 112.148,Z 997.891,A -85,B 0,C 180,E1 5823.513,E2 5823.513} C_VEL
LIN {X 0,Y 112.091,Z 998.675,A -85,B 0,C 180,E1 5816.409,E2 5816.409} C_VEL
LIN {X 0,Y 112.497,Z 998.899,A -85,B 0,C 180,E1 5808.179,E2 5808.179} C_VEL
LIN {X 0,Y 114.277,Z 998.299,A -85,B 0,C 180,E1 5798.84,E2 5798.84} C_VEL
LIN {X 0,Y 119.975,Z 996.056,A -85,B 0,C 180,E1 5786.885,E2 5786.885} C_VEL
LIN {X 0,Y 128.637,Z 992.545,A -85,B 0,C 180,E1 5777.018,E2 5777.018} C_VEL
LIN {X 0,Y 142.176,Z 986.811,A -85,B 0,C 180,E1 5767.372,E2 5767.372} C_VEL
LIN {X 0,Y 157.999,Z 979.693,A -85,B 0,C 180,E1 5759.828,E2 5759.828} C_VEL
LIN {X 0,Y 176.066,Z 970.599,A -85,B 0,C 180,E1 5753.678,E2 5753.678} C_VEL
LIN {X 0,Y 196.554,Z 959.217,A -85,B 0,C 180,E1 5748.558,E2 5748.558} C_VEL
LIN {X 0,Y 215.496,Z 947.564,A -85,B 0,C 180,E1 5744.911,E2 5744.911} C_VEL
LIN {X 0,Y 196.273,Z 960.158,A -85,B 0,C 180,E1 5741.374,E2 5741.374} C_VEL
LIN {X 0,Y 176.525,Z 972.08,A -85,B 0,C 180,E1 5736.592,E2 5736.592} C_VEL
LIN {X 0,Y 159.098,Z 981.742,A -85,B 0,C 180,E1 5730.89,E2 5730.89} C_VEL
LIN {X 0,Y 142.388,Z 990.408,A -85,B 0,C 180,E1 5723.194,E2 5723.194} C_VEL
LIN {X 0,Y 139.45,Z 991.898,A -85,B 0,C 180,E1 5721.492,E2 5721.492} C_VEL
LIN {X 0,Y 134.579,Z 994.066,A -85,B 0,C 180,E1 5719.127,E2 5719.127} C_VEL
LIN {X 0,Y 119.549,Z 999.159,A -85,B 0,C 180,E1 5712.733,E2 5712.733} C_VEL
LIN {X 0,Y 116.112,Z 1000.39,A -85,B 0,C 180,E1 5710.02,E2 5710.02} C_VEL
LIN {X 0,Y 108.214,Z 1004.062,A -85,B 0,C 180,E1 5698.128,E2 5698.128} C_VEL
LIN {X 0,Y 104.66,Z 1006.176,A -85,B 0,C 180,E1 5686.098,E2 5686.098} C_VEL
LIN {X 0,Y 104.051,Z 1006.721,A -85,B 0,C 180,E1 5676.082,E2 5676.082} C_VEL
LIN {X 0,Y 104.107,Z 1006.522,A -85,B 0,C 180,E1 5668.914,E2 5668.914} C_VEL
LIN {X 0,Y 104.119,Z 1005.497,A -85,B 0,C 180,E1 5660.619,E2 5660.619} C_VEL
LIN {X 0,Y 105.404,Z 1003.004,A -85,B 0,C 180,E1 5650.048,E2 5650.048} C_VEL
LIN {X 0,Y 109.164,Z 999.304,A -85,B 0,C 180,E1 5639.768,E2 5639.768} C_VEL
LIN {X 0,Y 116.84,Z 993.334,A -85,B 0,C 180,E1 5628.801,E2 5628.801} C_VEL
LIN {X 0,Y 126.702,Z 986.305,A -85,B 0,C 180,E1 5620.072,E2 5620.072} C_VEL
LIN {X 0,Y 139.516,Z 977.087,A -85,B 0,C 180,E1 5612.281,E2 5612.281} C_VEL
LIN {X 0,Y 153.587,Z 966.567,A -85,B 0,C 180,E1 5606.08,E2 5606.08} C_VEL
LIN {X 0,Y 168.281,Z 954.555,A -85,B 0,C 180,E1 5601.15,E2 5601.15} C_VEL
LIN {X 0,Y 183.98,Z 940.627,A -85,B 0,C 180,E1 5596.998,E2 5596.998} C_VEL
LIN {X 0,Y 198.7,Z 926.07,A -85,B 0,C 180,E1 5593.83,E2 5593.83} C_VEL
LIN {X 0,Y 213.939,Z 909.281,A -85,B 0,C 180,E1 5591.1,E2 5591.1} C_VEL
LIN {X 0,Y 228.2,Z 891.709,A -85,B 0,C 180,E1 5588.93,E2 5588.93} C_VEL
LIN {X 0,Y 241.33,Z 873.187,A -85,B 0,C 180,E1 5587.192,E2 5587.192} C_VEL
LIN {X 0,Y 253.918,Z 853.106,A -85,B 0,C 180,E1 5585.725,E2 5585.725} C_VEL
LIN {X 0,Y 264.776,Z 833.055,A -85,B 0,C 180,E1 5584.59,E2 5584.59} C_VEL
LIN {X 0,Y 275.158,Z 810.573,A -85,B 0,C 180,E1 5583.612,E2 5583.612} C_VEL
LIN {X 0,Y 283.78,Z 788.366,A -85,B 0,C 180,E1 5582.871,E2 5582.871} C_VEL
LIN {X 0,Y 290.918,Z 765.312,A -85,B 0,C 180,E1 5582.312,E2 5582.312} C_VEL
LIN {X 0,Y 296.854,Z 740.285,A -85,B 0,C 180,E1 5581.834,E2 5581.834} C_VEL
LIN {X 0,Y 300.778,Z 716.37,A -85,B 0,C 180,E1 5581.421,E2 5581.421} C_VEL
LIN {X 0,Y 311.424,Z 631.697,A -85,B 0,C 180,E1 5580.045,E2 5580.045} C_VEL
LIN {X 0,Y 308.84,Z 627.181,A -85,B 0,C 180,E1 5576.659,E2 5576.659} C_VEL
LIN {X 0,Y 306.735,Z 623.279,A -85,B 0,C 180,E1 5572.884,E2 5572.884} C_VEL
LIN {X 0,Y 304.813,Z 619.124,A -85,B 0,C 180,E1 5566.127,E2 5566.127} C_VEL
LIN {X 0,Y 304.687,Z 618.705,A -85,B 0,C 180,E1 5562.821,E2 5562.821} C_VEL
LIN {X 0,Y 304.849,Z 619.248,A -85,B 0,C 180,E1 5560.853,E2 5560.853} C_VEL
LIN {X 0,Y 306.87,Z 623.396,A -85,B 0,C 180,E1 5554.048,E2 5554.048} C_VEL
LIN {X 0,Y 309.67,Z 628.539,A -85,B 0,C 180,E1 5549.433,E2 5549.433} C_VEL
LIN {X 0,Y 311.175,Z 631.426,A -85,B 0,C 180,E1 5547.462,E2 5547.462} C_VEL
LIN {X 0,Y 299.209,Z 723.976,A -85,B 0,C 180,E1 5546,E2 5546} C_VEL
LIN {X 0,Y 294.388,Z 747.694,A -85,B 0,C 180,E1 5545.556,E2 5545.556} C_VEL
LIN {X 0,Y 288.397,Z 770.071,A -85,B 0,C 180,E1 5545.006,E2 5545.006} C_VEL
LIN {X 0,Y 280.99,Z 791.732,A -85,B 0,C 180,E1 5544.309,E2 5544.309} C_VEL
LIN {X 0,Y 271.183,Z 815.388,A -85,B 0,C 180,E1 5543.323,E2 5543.323} C_VEL
LIN {X 0,Y 260.688,Z 836.716,A -85,B 0,C 180,E1 5542.183,E2 5542.183} C_VEL
LIN {X 0,Y 248.962,Z 856.866,A -85,B 0,C 180,E1 5540.803,E2 5540.803} C_VEL
LIN {X 0,Y 235.24,Z 877.438,A -85,B 0,C 180,E1 5538.994,E2 5538.994} C_VEL
LIN {X 0,Y 222.008,Z 894.876,A -85,B 0,C 180,E1 5537.021,E2 5537.021} C_VEL
LIN {X 0,Y 207.839,Z 911.316,A -85,B 0,C 180,E1 5534.605,E2 5534.605} C_VEL
LIN {X 0,Y 193.599,Z 926.246,A -85,B 0,C 180,E1 5531.765,E2 5531.765} C_VEL
LIN {X 0,Y 178.209,Z 940.527,A -85,B 0,C 180,E1 5528.097,E2 5528.097} C_VEL
LIN {X 0,Y 162.072,Z 954.115,A -85,B 0,C 180,E1 5523.29,E2 5523.29} C_VEL
LIN {X 0,Y 148.473,Z 964.592,A -85,B 0,C 180,E1 5518.113,E2 5518.113} C_VEL
LIN {X 0,Y 134.876,Z 974.319,A -85,B 0,C 180,E1 5511.287,E2 5511.287} C_VEL
LIN {X 0,Y 123.184,Z 982.431,A -85,B 0,C 180,E1 5503.083,E2 5503.083} C_VEL
LIN {X 0,Y 114.024,Z 988.728,A -85,B 0,C 180,E1 5493.506,E2 5493.506} C_VEL
LIN {X 0,Y 107.79,Z 993.662,A -85,B 0,C 180,E1 5482.524,E2 5482.524} C_VEL
LIN {X 0,Y 104.855,Z 996.697,A -85,B 0,C 180,E1 5471.644,E2 5471.644} C_VEL
LIN {X 0,Y 104.143,Z 998.218,A -85,B 0,C 180,E1 5463.162,E2 5463.162} C_VEL
LIN {X 0,Y 104.102,Z 998.985,A -85,B 0,C 180,E1 5455.693,E2 5455.693} C_VEL
LIN {X 0,Y 104.577,Z 999.23,A -85,B 0,C 180,E1 5447.23,E2 5447.23} C_VEL
LIN {X 0,Y 106.707,Z 998.677,A -85,B 0,C 180,E1 5437.186,E2 5437.186} C_VEL
LIN {X 0,Y 112.729,Z 996.722,A -85,B 0,C 180,E1 5425.191,E2 5425.191} C_VEL
LIN {X 0,Y 122.807,Z 993.095,A -85,B 0,C 180,E1 5414.293,E2 5414.293} C_VEL
LIN {X 0,Y 137.438,Z 987.51,A -85,B 0,C 180,E1 5404.564,E2 5404.564} C_VEL
LIN {X 0,Y 154.438,Z 980.417,A -85,B 0,C 180,E1 5397.032,E2 5397.032} C_VEL
LIN {X 0,Y 173.045,Z 971.647,A -85,B 0,C 180,E1 5391.175,E2 5391.175} C_VEL
LIN {X 0,Y 193.061,Z 961.22,A -85,B 0,C 180,E1 5386.524,E2 5386.524} C_VEL
LIN {X 0,Y 201.075,Z 956.675,A -85,B 0,C 180,E1 5384.982,E2 5384.982} C_VEL
LIN {X 0,Y 181.774,Z 968.046,A -85,B 0,C 180,E1 5381.121,E2 5381.121} C_VEL
LIN {X 0,Y 161.375,Z 978.999,A -85,B 0,C 180,E1 5375.633,E2 5375.633} C_VEL
LIN {X 0,Y 142.932,Z 988.147,A -85,B 0,C 180,E1 5368.604,E2 5368.604} C_VEL
LIN {X 0,Y 127.172,Z 995.33,A -85,B 0,C 180,E1 5359.713,E2 5359.713} C_VEL
LIN {X 0,Y 116.112,Z 1000.39,A -85,B 0,C 180,E1 5350.02,E2 5350.02} C_VEL
LIN {X 0,Y 112.301,Z 1001.683,A -85,B 0,C 180,E1 5346.684,E2 5346.684} C_VEL
LIN {X 0,Y 103.145,Z 1003.908,A -85,B 0,C 180,E1 5340.004,E2 5340.004} C_VEL
LIN {X 0,Y 98.993,Z 1004.884,A -85,B 0,C 180,E1 5335.193,E2 5335.193} C_VEL
LIN {X 0,Y 98.323,Z 1005.098,A -85,B 0,C 180,E1 5333.627,E2 5333.627} C_VEL
LIN {X 0,Y 96.229,Z 1006.215,A -85,B 0,C 180,E1 5322.402,E2 5322.402} C_VEL
LIN {X 0,Y 96.07,Z 1006.331,A -85,B 0,C 180,E1 5313.596,E2 5313.596} C_VEL
LIN {X 0,Y 96.093,Z 1005.949,A -85,B 0,C 180,E1 5307.034,E2 5307.034} C_VEL
LIN {X 0,Y 96.195,Z 1004.826,A -85,B 0,C 180,E1 5298.626,E2 5298.626} C_VEL
LIN {X 0,Y 97.735,Z 1002.504,A -85,B 0,C 180,E1 5288.407,E2 5288.407} C_VEL
LIN {X 0,Y 102.387,Z 998.519,A -85,B 0,C 180,E1 5276.866,E2 5276.866} C_VEL
LIN {X 0,Y 110.678,Z 992.63,A -85,B 0,C 180,E1 5265.945,E2 5265.945} C_VEL
LIN {X 0,Y 122.057,Z 985.152,A -85,B 0,C 180,E1 5256.626,E2 5256.626} C_VEL
LIN {X 0,Y 135.894,Z 975.677,A -85,B 0,C 180,E1 5248.916,E2 5248.916} C_VEL
LIN {X 0,Y 150.836,Z 964.873,A -85,B 0,C 180,E1 5242.899,E2 5242.899} C_VEL
LIN {X 0,Y 165.959,Z 952.893,A -85,B 0,C 180,E1 5238.256,E2 5238.256} C_VEL
LIN {X 0,Y 182.552,Z 938.358,A -85,B 0,C 180,E1 5234.241,E2 5234.241} C_VEL
LIN {X 0,Y 198.206,Z 923.157,A -85,B 0,C 180,E1 5231.187,E2 5231.187} C_VEL
LIN {X 0,Y 213.401,Z 906.396,A -85,B 0,C 180,E1 5228.716,E2 5228.716} C_VEL
LIN {X 0,Y 228.463,Z 887.686,A -85,B 0,C 180,E1 5226.634,E2 5226.634} C_VEL
LIN {X 0,Y 240.899,Z 870.146,A -85,B 0,C 180,E1 5225.138,E2 5225.138} C_VEL
LIN {X 0,Y 253.485,Z 849.823,A -85,B 0,C 180,E1 5223.795,E2 5223.795} C_VEL
LIN {X 0,Y 264.726,Z 828.957,A -85,B 0,C 180,E1 5222.725,E2 5222.725} C_VEL
LIN {X 0,Y 274.534,Z 807.248,A -85,B 0,C 180,E1 5221.878,E2 5221.878} C_VEL
LIN {X 0,Y 283.483,Z 783.468,A -85,B 0,C 180,E1 5221.173,E2 5221.173} C_VEL
LIN {X 0,Y 290.557,Z 760.194,A -85,B 0,C 180,E1 5220.672,E2 5220.672} C_VEL
LIN {X 0,Y 295.82,Z 736.674,A -85,B 0,C 180,E1 5220.26,E2 5220.26} C_VEL
LIN {X 0,Y 300.373,Z 706.529,A -85,B 0,C 180,E1 5219.772,E2 5219.772} C_VEL
LIN {X 0,Y 309.167,Z 637.98,A -85,B 0,C 180,E1 5218.702,E2 5218.702} C_VEL
LIN {X 0,Y 307.434,Z 634.825,A -85,B 0,C 180,E1 5216.27,E2 5216.27} C_VEL
LIN {X 0,Y 305.465,Z 631.081,A -85,B 0,C 180,E1 5212.599,E2 5212.599} C_VEL
LIN {X 0,Y 303.604,Z 626.682,A -85,B 0,C 180,E1 5205.115,E2 5205.115} C_VEL
LIN {X 0,Y 303.682,Z 626.85,A -85,B 0,C 180,E1 5201.375,E2 5201.375} C_VEL
LIN {X 0,Y 305.366,Z 630.955,A -85,B 0,C 180,E1 5194.807,E2 5194.807} C_VEL
LIN {X 0,Y 306.068,Z 632.29,A -85,B 0,C 180,E1 5193.308,E2 5193.308} C_VEL
LIN {X 0,Y 308.368,Z 636.429,A -85,B 0,C 180,E1 5189.614,E2 5189.614} C_VEL
LIN {X 0,Y 308.905,Z 637.777,A -85,B 0,C 180,E1 5188.821,E2 5188.821} C_VEL
LIN {X 0,Y 297.464,Z 724.53,A -85,B 0,C 180,E1 5187.496,E2 5187.496} C_VEL
LIN {X 0,Y 292.564,Z 748.21,A -85,B 0,C 180,E1 5187.073,E2 5187.073} C_VEL
LIN {X 0,Y 286.386,Z 770.873,A -85,B 0,C 180,E1 5186.543,E2 5186.543} C_VEL
LIN {X 0,Y 278.931,Z 792.389,A -85,B 0,C 180,E1 5185.886,E2 5185.886} C_VEL
LIN {X 0,Y 269.2,Z 815.564,A -85,B 0,C 180,E1 5184.97,E2 5184.97} C_VEL
LIN {X 0,Y 258.605,Z 836.852,A -85,B 0,C 180,E1 5183.895,E2 5183.895} C_VEL
LIN {X 0,Y 246.698,Z 857.064,A -85,B 0,C 180,E1 5182.584,E2 5182.584} C_VEL
LIN {X 0,Y 233.114,Z 877.163,A -85,B 0,C 180,E1 5180.913,E2 5180.913} C_VEL
LIN {X 0,Y 219.667,Z 894.59,A -85,B 0,C 180,E1 5179.046,E2 5179.046} C_VEL
LIN {X 0,Y 204.763,Z 911.571,A -85,B 0,C 180,E1 5176.67,E2 5176.67} C_VEL
LIN {X 0,Y 190.165,Z 926.524,A -85,B 0,C 180,E1 5173.937,E2 5173.937} C_VEL
LIN {X 0,Y 174.325,Z 940.837,A -85,B 0,C 180,E1 5170.387,E2 5170.387} C_VEL
LIN {X 0,Y 157.618,Z 954.451,A -85,B 0,C 180,E1 5165.691,E2 5165.691} C_VEL
LIN {X 0,Y 143.44,Z 964.939,A -85,B 0,C 180,E1 5160.574,E2 5160.574} C_VEL
LIN {X 0,Y 129.135,Z 974.657,A -85,B 0,C 180,E1 5153.729,E2 5153.729} C_VEL
LIN {X 0,Y 116.746,Z 982.738,A -85,B 0,C 180,E1 5145.383,E2 5145.383} C_VEL
LIN {X 0,Y 106.847,Z 989.059,A -85,B 0,C 180,E1 5135.355,E2 5135.355} C_VEL
LIN {X 0,Y 100.067,Z 993.99,A -85,B 0,C 180,E1 5123.675,E2 5123.675} C_VEL
LIN {X 0,Y 96.849,Z 997.053,A -85,B 0,C 180,E1 5111.774,E2 5111.774} C_VEL
LIN {X 0,Y 96.14,Z 998.536,A -85,B 0,C 180,E1 5102.751,E2 5102.751} C_VEL
LIN {X 0,Y 96.117,Z 999.28,A -85,B 0,C 180,E1 5095.083,E2 5095.083} C_VEL
LIN {X 0,Y 96.69,Z 999.564,A -85,B 0,C 180,E1 5086.125,E2 5086.125} C_VEL
LIN {X 0,Y 99.334,Z 999.04,A -85,B 0,C 180,E1 5075.014,E2 5075.014} C_VEL
LIN {X 0,Y 106.659,Z 997.026,A -85,B 0,C 180,E1 5061.833,E2 5061.833} C_VEL
LIN {X 0,Y 118.062,Z 993.415,A -85,B 0,C 180,E1 5050.71,E2 5050.71} C_VEL
LIN {X 0,Y 134.513,Z 987.682,A -85,B 0,C 180,E1 5040.853,E2 5040.853} C_VEL
LIN {X 0,Y 152.966,Z 980.512,A -85,B 0,C 180,E1 5033.556,E2 5033.556} C_VEL
LIN {X 0,Y 172.877,Z 971.579,A -85,B 0,C 180,E1 5027.984,E2 5027.984} C_VEL
LIN {X 0,Y 186.341,Z 964.977,A -85,B 0,C 180,E1 5025.003,E2 5025.003} C_VEL
LIN {X 0,Y 165.59,Z 975.901,A -85,B 0,C 180,E1 5020.403,E2 5020.403} C_VEL
LIN {X 0,Y 145.495,Z 985.346,A -85,B 0,C 180,E1 5014.21,E2 5014.21} C_VEL
LIN {X 0,Y 127,Z 993.36,A -85,B 0,C 180,E1 5005.775,E2 5005.775} C_VEL
LIN {X 0,Y 112.96,Z 999.048,A -85,B 0,C 180,E1 4995.822,E2 4995.822} C_VEL
LIN {X 0,Y 102.348,Z 1003.33,A -85,B 0,C 180,E1 4982.847,E2 4982.847} C_VEL
LIN {X 0,Y 98.323,Z 1005.098,A -85,B 0,C 180,E1 4973.627,E2 4973.627} C_VEL
LIN {X 0,Y 96.204,Z 1005.724,A -85,B 0,C 180,E1 4969.24,E2 4969.24} C_VEL
LIN {X 0,Y 91.357,Z 1006.118,A -85,B 0,C 180,E1 4961.942,E2 4961.942} C_VEL
LIN {X 0,Y 88.215,Z 1006.019,A -85,B 0,C 180,E1 4954.265,E2 4954.265} C_VEL
LIN {X 0,Y 88.094,Z 1005.972,A -85,B 0,C 180,E1 4952.434,E2 4952.434} C_VEL
LIN {X 0,Y 88.087,Z 1005.372,A -85,B 0,C 180,E1 4944.807,E2 4944.807} C_VEL
LIN {X 0,Y 88.501,Z 1003.915,A -85,B 0,C 180,E1 4934.957,E2 4934.957} C_VEL
LIN {X 0,Y 91.874,Z 1000.566,A -85,B 0,C 180,E1 4921.41,E2 4921.41} C_VEL
LIN {X 0,Y 98.858,Z 995.673,A -85,B 0,C 180,E1 4909.334,E2 4909.334} C_VEL
LIN {X 0,Y 109.8,Z 988.878,A -85,B 0,C 180,E1 4898.476,E2 4898.476} C_VEL
LIN {X 0,Y 122.614,Z 980.837,A -85,B 0,C 180,E1 4890.216,E2 4890.216} C_VEL
LIN {X 0,Y 138.14,Z 970.54,A -85,B 0,C 180,E1 4883.219,E2 4883.219} C_VEL
LIN {X 0,Y 153.545,Z 959.436,A -85,B 0,C 180,E1 4878.099,E2 4878.099} C_VEL
LIN {X 0,Y 169.92,Z 946.302,A -85,B 0,C 180,E1 4873.9,E2 4873.9} C_VEL
LIN {X 0,Y 186.115,Z 931.906,A -85,B 0,C 180,E1 4870.596,E2 4870.596} C_VEL
LIN {X 0,Y 201.709,Z 916.188,A -85,B 0,C 180,E1 4867.977,E2 4867.977} C_VEL
LIN {X 0,Y 217.529,Z 898.238,A -85,B 0,C 180,E1 4865.748,E2 4865.748} C_VEL
LIN {X 0,Y 231.515,Z 880.274,A -85,B 0,C 180,E1 4864.065,E2 4864.065} C_VEL
LIN {X 0,Y 244.697,Z 860.779,A -85,B 0,C 180,E1 4862.675,E2 4862.675} C_VEL
LIN {X 0,Y 256.617,Z 840.671,A -85,B 0,C 180,E1 4861.562,E2 4861.562} C_VEL
LIN {X 0,Y 266.946,Z 820.255,A -85,B 0,C 180,E1 4860.696,E2 4860.696} C_VEL
LIN {X 0,Y 276.925,Z 796.851,A -85,B 0,C 180,E1 4859.936,E2 4859.936} C_VEL
LIN {X 0,Y 284.488,Z 775.408,A -85,B 0,C 180,E1 4859.415,E2 4859.415} C_VEL
LIN {X 0,Y 290.933,Z 752.038,A -85,B 0,C 180,E1 4858.988,E2 4858.988} C_VEL
LIN {X 0,Y 295.843,Z 728.015,A -85,B 0,C 180,E1 4858.595,E2 4858.595} C_VEL
LIN {X 0,Y 306.982,Z 644.209,A -85,B 0,C 180,E1 4857.339,E2 4857.339} C_VEL
LIN {X 0,Y 304.384,Z 639.078,A -85,B 0,C 180,E1 4852.705,E2 4852.705} C_VEL
LIN {X 0,Y 302.517,Z 634.905,A -85,B 0,C 180,E1 4845.842,E2 4845.842} C_VEL
LIN {X 0,Y 302.46,Z 634.578,A -85,B 0,C 180,E1 4842.294,E2 4842.294} C_VEL
LIN {X 0,Y 302.578,Z 635.344,A -85,B 0,C 180,E1 4840.704,E2 4840.704} C_VEL
LIN {X 0,Y 304.632,Z 639.671,A -85,B 0,C 180,E1 4833.907,E2 4833.907} C_VEL
LIN {X 0,Y 306.778,Z 643.798,A -85,B 0,C 180,E1 4830.202,E2 4830.202} C_VEL
LIN {X 0,Y 295.949,Z 724.789,A -85,B 0,C 180,E1 4829.012,E2 4829.012} C_VEL
LIN {X 0,Y 290.981,Z 748.54,A -85,B 0,C 180,E1 4828.612,E2 4828.612} C_VEL
LIN {X 0,Y 284.745,Z 771.165,A -85,B 0,C 180,E1 4828.114,E2 4828.114} C_VEL
LIN {X 0,Y 277.333,Z 792.323,A -85,B 0,C 180,E1 4827.507,E2 4827.507} C_VEL
LIN {X 0,Y 267.444,Z 815.639,A -85,B 0,C 180,E1 4826.642,E2 4826.642} C_VEL
LIN {X 0,Y 257.037,Z 836.318,A -85,B 0,C 180,E1 4825.663,E2 4825.663} C_VEL
LIN {X 0,Y 245.129,Z 856.391,A -85,B 0,C 180,E1 4824.45,E2 4824.45} C_VEL
LIN {X 0,Y 231.776,Z 876.062,A -85,B 0,C 180,E1 4822.933,E2 4822.933} C_VEL
LIN {X 0,Y 218.111,Z 893.598,A -85,B 0,C 180,E1 4821.184,E2 4821.184} C_VEL
LIN {X 0,Y 202.847,Z 910.862,A -85,B 0,C 180,E1 4818.938,E2 4818.938} C_VEL
LIN {X 0,Y 187.88,Z 925.938,A -85,B 0,C 180,E1 4816.352,E2 4816.352} C_VEL
LIN {X 0,Y 172.418,Z 939.688,A -85,B 0,C 180,E1 4813.165,E2 4813.165} C_VEL
LIN {X 0,Y 156.679,Z 952.386,A -85,B 0,C 180,E1 4809.167,E2 4809.167} C_VEL
LIN {X 0,Y 140.95,Z 963.652,A -85,B 0,C 180,E1 4804.069,E2 4804.069} C_VEL
LIN {X 0,Y 125.697,Z 973.719,A -85,B 0,C 180,E1 4797.46,E2 4797.46} C_VEL
LIN {X 0,Y 112.803,Z 981.596,A -85,B 0,C 180,E1 4789.669,E2 4789.669} C_VEL
LIN {X 0,Y 100.687,Z 988.851,A -85,B 0,C 180,E1 4778.551,E2 4778.551} C_VEL
LIN {X 0,Y 93.511,Z 993.448,A -85,B 0,C 180,E1 4767.533,E2 4767.533} C_VEL
LIN {X 0,Y 89.251,Z 996.955,A -85,B 0,C 180,E1 4754.386,E2 4754.386} C_VEL
LIN {X 0,Y 88.162,Z 998.697,A -85,B 0,C 180,E1 4743.635,E2 4743.635} C_VEL
LIN {X 0,Y 88.13,Z 999.562,A -85,B 0,C 180,E1 4734.628,E2 4734.628} C_VEL
LIN {X 0,Y 88.978,Z 999.887,A -85,B 0,C 180,E1 4723.991,E2 4723.991} C_VEL
LIN {X 0,Y 92.569,Z 999.321,A -85,B 0,C 180,E1 4711.401,E2 4711.401} C_VEL
LIN {X 0,Y 101.847,Z 997.103,A -85,B 0,C 180,E1 4697.13,E2 4697.13} C_VEL
LIN {X 0,Y 115.087,Z 993.403,A -85,B 0,C 180,E1 4685.986,E2 4685.986} C_VEL
LIN {X 0,Y 132.235,Z 987.875,A -85,B 0,C 180,E1 4676.967,E2 4676.967} C_VEL
LIN {X 0,Y 151.711,Z 980.784,A -85,B 0,C 180,E1 4670.135,E2 4670.135} C_VEL
LIN {X 0,Y 171.797,Z 972.241,A -85,B 0,C 180,E1 4665.069,E2 4665.069} C_VEL
LIN {X 0,Y 151.088,Z 981.928,A -85,B 0,C 180,E1 4660.027,E2 4660.027} C_VEL
LIN {X 0,Y 131.205,Z 990.127,A -85,B 0,C 180,E1 4653.097,E2 4653.097} C_VEL
LIN {X 0,Y 113.242,Z 996.931,A -85,B 0,C 180,E1 4643.483,E2 4643.483} C_VEL
LIN {X 0,Y 100.194,Z 1001.549,A -85,B 0,C 180,E1 4631.978,E2 4631.978} C_VEL
LIN {X 0,Y 91.435,Z 1004.663,A -85,B 0,C 180,E1 4617.358,E2 4617.358} C_VEL
LIN {X 0,Y 88.477,Z 1005.848,A -85,B 0,C 180,E1 4605.082,E2 4605.082} C_VEL
LIN {X 0,Y 88.065,Z 1006.022,A -85,B 0,C 180,E1 4595.228,E2 4595.228} C_VEL
LIN {X 0,Y 88.094,Z 1005.972,A -85,B 0,C 180,E1 4592.434,E2 4592.434} C_VEL
LIN {X 0,Y 87.352,Z 1005.754,A -85,B 0,C 180,E1 4588.142,E2 4588.142} C_VEL
LIN {X 0,Y 84.881,Z 1005.115,A -85,B 0,C 180,E1 4582.443,E2 4582.443} C_VEL
LIN {X 0,Y 81.27,Z 1003.209,A -85,B 0,C 180,E1 4571.758,E2 4571.758} C_VEL
LIN {X 0,Y 81.509,Z 1002.507,A -85,B 0,C 180,E1 4568.59,E2 4568.59} C_VEL
LIN {X 0,Y 86.313,Z 998.879,A -85,B 0,C 180,E1 4555.438,E2 4555.438} C_VEL
LIN {X 0,Y 95.994,Z 993.108,A -85,B 0,C 180,E1 4542.335,E2 4542.335} C_VEL
LIN {X 0,Y 108.026,Z 986.175,A -85,B 0,C 180,E1 4532.649,E2 4532.649} C_VEL
LIN {X 0,Y 123.878,Z 976.657,A -85,B 0,C 180,E1 4524.243,E2 4524.243} C_VEL
LIN {X 0,Y 139.693,Z 966.348,A -85,B 0,C 180,E1 4518.355,E2 4518.355} C_VEL
LIN {X 0,Y 156.551,Z 954.061,A -85,B 0,C 180,E1 4513.668,E2 4513.668} C_VEL
LIN {X 0,Y 173.576,Z 940.276,A -85,B 0,C 180,E1 4509.992,E2 4509.992} C_VEL
LIN {X 0,Y 189.448,Z 925.732,A -85,B 0,C 180,E1 4507.232,E2 4507.232} C_VEL
LIN {X 0,Y 206.402,Z 908.204,A -85,B 0,C 180,E1 4504.806,E2 4504.806} C_VEL
LIN {X 0,Y 221.241,Z 890.826,A -85,B 0,C 180,E1 4503.016,E2 4503.016} C_VEL
LIN {X 0,Y 235.021,Z 872.214,A -85,B 0,C 180,E1 4501.573,E2 4501.573} C_VEL
LIN {X 0,Y 248.434,Z 851.542,A -85,B 0,C 180,E1 4500.344,E2 4500.344} C_VEL
LIN {X 0,Y 259.44,Z 831.862,A -85,B 0,C 180,E1 4499.443,E2 4499.443} C_VEL
LIN {X 0,Y 269.999,Z 809.638,A -85,B 0,C 180,E1 4498.664,E2 4498.664} C_VEL
LIN {X 0,Y 278.832,Z 787.536,A -85,B 0,C 180,E1 4498.073,E2 4498.073} C_VEL
LIN {X 0,Y 286.168,Z 764.509,A -85,B 0,C 180,E1 4497.63,E2 4497.63} C_VEL
LIN {X 0,Y 292.293,Z 739.387,A -85,B 0,C 180,E1 4497.237,E2 4497.237} C_VEL
LIN {X 0,Y 296.361,Z 715.481,A -85,B 0,C 180,E1 4496.877,E2 4496.877} C_VEL
LIN {X 0,Y 304.921,Z 650.533,A -85,B 0,C 180,E1 4495.927,E2 4495.927} C_VEL
LIN {X 0,Y 302.994,Z 646.778,A -85,B 0,C 180,E1 4492.224,E2 4492.224} C_VEL
LIN {X 0,Y 301.33,Z 642.504,A -85,B 0,C 180,E1 4484.897,E2 4484.897} C_VEL
LIN {X 0,Y 301.396,Z 642.804,A -85,B 0,C 180,E1 4481.429,E2 4481.429} C_VEL
LIN {X 0,Y 303.35,Z 647.403,A -85,B 0,C 180,E1 4474.209,E2 4474.209} C_VEL
LIN {X 0,Y 304.724,Z 650.281,A -85,B 0,C 180,E1 4471.594,E2 4471.594} C_VEL
LIN {X 0,Y 294.488,Z 725.408,A -85,B 0,C 180,E1 4470.535,E2 4470.535} C_VEL
LIN {X 0,Y 289.433,Z 749.15,A -85,B 0,C 180,E1 4470.158,E2 4470.158} C_VEL
LIN {X 0,Y 282.891,Z 772.401,A -85,B 0,C 180,E1 4469.673,E2 4469.673} C_VEL
LIN {X 0,Y 275.504,Z 793.201,A -85,B 0,C 180,E1 4469.113,E2 4469.113} C_VEL
LIN {X 0,Y 265.534,Z 816.358,A -85,B 0,C 180,E1 4468.306,E2 4468.306} C_VEL
LIN {X 0,Y 254.606,Z 837.752,A -85,B 0,C 180,E1 4467.351,E2 4467.351} C_VEL
LIN {X 0,Y 242.416,Z 857.873,A -85,B 0,C 180,E1 4466.197,E2 4466.197} C_VEL
LIN {X 0,Y 227.941,Z 878.596,A -85,B 0,C 180,E1 4464.661,E2 4464.661} C_VEL
LIN {X 0,Y 213.61,Z 896.499,A -85,B 0,C 180,E1 4462.932,E2 4462.932} C_VEL
LIN {X 0,Y 198.53,Z 912.878,A -85,B 0,C 180,E1 4460.844,E2 4460.844} C_VEL
LIN {X 0,Y 182.371,Z 928.536,A -85,B 0,C 180,E1 4458.198,E2 4458.198} C_VEL
LIN {X 0,Y 166.574,Z 942.036,A -85,B 0,C 180,E1 4455.081,E2 4455.081} C_VEL
LIN {X 0,Y 148.773,Z 955.57,A -85,B 0,C 180,E1 4450.671,E2 4450.671} C_VEL
LIN {X 0,Y 132.378,Z 966.77,A -85,B 0,C 180,E1 4445.338,E2 4445.338} C_VEL
LIN {X 0,Y 117.032,Z 976.094,A -85,B 0,C 180,E1 4438.567,E2 4438.567} C_VEL
LIN {X 0,Y 102.613,Z 984.329,A -85,B 0,C 180,E1 4429.331,E2 4429.331} C_VEL
LIN {X 0,Y 91.964,Z 990.219,A -85,B 0,C 180,E1 4418.738,E2 4418.738} C_VEL
LIN {X 0,Y 83.944,Z 995.127,A -85,B 0,C 180,E1 4404.514,E2 4404.514} C_VEL
LIN {X 0,Y 80.817,Z 997.77,A -85,B 0,C 180,E1 4391.964,E2 4391.964} C_VEL
LIN {X 0,Y 80.136,Z 999.164,A -85,B 0,C 180,E1 4381.677,E2 4381.677} C_VEL
LIN {X 0,Y 80.196,Z 999.923,A -85,B 0,C 180,E1 4372.322,E2 4372.322} C_VEL
LIN {X 0,Y 81.566,Z 1000.204,A -85,B 0,C 180,E1 4360.509,E2 4360.509} C_VEL
LIN {X 0,Y 86.383,Z 999.585,A -85,B 0,C 180,E1 4346.837,E2 4346.837} C_VEL
LIN {X 0,Y 97.292,Z 997.319,A -85,B 0,C 180,E1 4332.437,E2 4332.437} C_VEL
LIN {X 0,Y 112.069,Z 993.637,A -85,B 0,C 180,E1 4321.535,E2 4321.535} C_VEL
LIN {X 0,Y 131.035,Z 987.966,A -85,B 0,C 180,E1 4312.806,E2 4312.806} C_VEL
LIN {X 0,Y 151.214,Z 981.026,A -85,B 0,C 180,E1 4306.62,E2 4306.62} C_VEL
LIN {X 0,Y 157.103,Z 978.702,A -85,B 0,C 180,E1 4305.122,E2 4305.122} C_VEL
LIN {X 0,Y 135.648,Z 987.468,A -85,B 0,C 180,E1 4299.281,E2 4299.281} C_VEL
LIN {X 0,Y 116.217,Z 994.419,A -85,B 0,C 180,E1 4291.37,E2 4291.37} C_VEL
LIN {X 0,Y 98.494,Z 1000.136,A -85,B 0,C 180,E1 4279.605,E2 4279.605} C_VEL
LIN {X 0,Y 87.127,Z 1003.616,A -85,B 0,C 180,E1 4265.842,E2 4265.842} C_VEL
LIN {X 0,Y 81.236,Z 1005.379,A -85,B 0,C 180,E1 4250.178,E2 4250.178} C_VEL
LIN {X 0,Y 80.066,Z 1005.717,A -85,B 0,C 180,E1 4237.914,E2 4237.914} C_VEL
LIN {X 0,Y 80.132,Z 1005.419,A -85,B 0,C 180,E1 4229.304,E2 4229.304} C_VEL
LIN {X 0,Y 80.148,Z 1004.499,A -85,B 0,C 180,E1 4219.961,E2 4219.961} C_VEL
LIN {X 0,Y 81.509,Z 1002.507,A -85,B 0,C 180,E1 4208.59,E2 4208.59} C_VEL
LIN {X 0,Y 81.969,Z 1001.256,A -85,B 0,C 180,E1 4203.239,E2 4203.239} C_VEL
LIN {X 0,Y 81.746,Z 998.393,A -85,B 0,C 180,E1 4192.823,E2 4192.823} C_VEL
LIN {X 0,Y 83.497,Z 996.218,A -85,B 0,C 180,E1 4186.5,E2 4186.5} C_VEL
LIN {X 0,Y 84.843,Z 995.37,A -85,B 0,C 180,E1 4184.486,E2 4184.486} C_VEL
LIN {X 0,Y 97.492,Z 988.716,A -85,B 0,C 180,E1 4172.789,E2 4172.789} C_VEL
LIN {X 0,Y 111.923,Z 980.724,A -85,B 0,C 180,E1 4164.363,E2 4164.363} C_VEL
LIN {X 0,Y 128.965,Z 970.529,A -85,B 0,C 180,E1 4157.565,E2 4157.565} C_VEL
LIN {X 0,Y 145.546,Z 959.466,A -85,B 0,C 180,E1 4152.765,E2 4152.765} C_VEL
LIN {X 0,Y 162.919,Z 946.415,A -85,B 0,C 180,E1 4148.928,E2 4148.928} C_VEL
LIN {X 0,Y 179.915,Z 932.106,A -85,B 0,C 180,E1 4145.962,E2 4145.962} C_VEL
LIN {X 0,Y 196.331,Z 916.263,A -85,B 0,C 180,E1 4143.621,E2 4143.621} C_VEL
LIN {X 0,Y 212.476,Z 898.674,A -85,B 0,C 180,E1 4141.698,E2 4141.698} C_VEL
LIN {X 0,Y 225.937,Z 881.987,A -85,B 0,C 180,E1 4140.325,E2 4140.325} C_VEL
LIN {X 0,Y 240.292,Z 861.624,A -85,B 0,C 180,E1 4139.046,E2 4139.046} C_VEL
LIN {X 0,Y 252.57,Z 841.619,A -85,B 0,C 180,E1 4138.085,E2 4138.085} C_VEL
LIN {X 0,Y 263.719,Z 820.103,A -85,B 0,C 180,E1 4137.304,E2 4137.304} C_VEL
LIN {X 0,Y 274.039,Z 796.358,A -85,B 0,C 180,E1 4136.653,E2 4136.653} C_VEL
LIN {X 0,Y 282.059,Z 773.951,A -85,B 0,C 180,E1 4136.202,E2 4136.202} C_VEL
LIN {X 0,Y 288.556,Z 750.434,A -85,B 0,C 180,E1 4135.844,E2 4135.844} C_VEL
LIN {X 0,Y 293.696,Z 724.884,A -85,B 0,C 180,E1 4135.477,E2 4135.477} C_VEL
LIN {X 0,Y 302.918,Z 657.185,A -85,B 0,C 180,E1 4134.539,E2 4134.539} C_VEL
LIN {X 0,Y 301.747,Z 654.608,A -85,B 0,C 180,E1 4132,E2 4132} C_VEL
LIN {X 0,Y 300.192,Z 650.411,A -85,B 0,C 180,E1 4124.744,E2 4124.744} C_VEL
LIN {X 0,Y 300.247,Z 650.704,A -85,B 0,C 180,E1 4121.556,E2 4121.556} C_VEL
LIN {X 0,Y 302.113,Z 655.254,A -85,B 0,C 180,E1 4114.411,E2 4114.411} C_VEL
LIN {X 0,Y 302.738,Z 657.039,A -85,B 0,C 180,E1 4113,E2 4113} C_VEL
LIN {X 0,Y 293.234,Z 725.886,A -85,B 0,C 180,E1 4112.072,E2 4112.072} C_VEL
LIN {X 0,Y 288.128,Z 749.58,A -85,B 0,C 180,E1 4111.721,E2 4111.721} C_VEL
LIN {X 0,Y 281.34,Z 773.35,A -85,B 0,C 180,E1 4111.259,E2 4111.259} C_VEL
LIN {X 0,Y 273.879,Z 794.064,A -85,B 0,C 180,E1 4110.738,E2 4110.738} C_VEL
LIN {X 0,Y 264.015,Z 816.654,A -85,B 0,C 180,E1 4110.006,E2 4110.006} C_VEL
LIN {X 0,Y 253.278,Z 837.475,A -85,B 0,C 180,E1 4109.147,E2 4109.147} C_VEL
LIN {X 0,Y 240.877,Z 857.762,A -85,B 0,C 180,E1 4108.073,E2 4108.073} C_VEL
LIN {X 0,Y 226.666,Z 877.947,A -85,B 0,C 180,E1 4106.696,E2 4106.696} C_VEL
LIN {X 0,Y 212.566,Z 895.412,A -85,B 0,C 180,E1 4105.15,E2 4105.15} C_VEL
LIN {X 0,Y 196.774,Z 912.482,A -85,B 0,C 180,E1 4103.158,E2 4103.158} C_VEL
LIN {X 0,Y 180.693,Z 927.913,A -85,B 0,C 180,E1 4100.761,E2 4100.761} C_VEL
LIN {X 0,Y 164.476,Z 941.514,A -85,B 0,C 180,E1 4097.856,E2 4097.856} C_VEL
LIN {X 0,Y 146.951,Z 954.61,A -85,B 0,C 180,E1 4093.932,E2 4093.932} C_VEL
LIN {X 0,Y 130.963,Z 965.207,A -85,B 0,C 180,E1 4089.305,E2 4089.305} C_VEL
LIN {X 0,Y 113.585,Z 975.508,A -85,B 0,C 180,E1 4082.46,E2 4082.46} C_VEL
LIN {X 0,Y 98.675,Z 983.626,A -85,B 0,C 180,E1 4073.893,E2 4073.893} C_VEL
LIN {X 0,Y 86.041,Z 990.047,A -85,B 0,C 180,E1 4062.532,E2 4062.532} C_VEL
LIN {X 0,Y 77.232,Z 994.905,A -85,B 0,C 180,E1 4048.497,E2 4048.497} C_VEL
LIN {X 0,Y 72.961,Z 997.94,A -85,B 0,C 180,E1 4033.254,E2 4033.254} C_VEL
LIN {X 0,Y 72.14,Z 999.384,A -85,B 0,C 180,E1 4021.863,E2 4021.863} C_VEL
LIN {X 0,Y 72.232,Z 1000.2,A -85,B 0,C 180,E1 4011.447,E2 4011.447} C_VEL
LIN {X 0,Y 73.943,Z 1000.546,A -85,B 0,C 180,E1 3998.316,E2 3998.316} C_VEL
LIN {X 0,Y 79.644,Z 999.995,A -85,B 0,C 180,E1 3983.546,E2 3983.546} C_VEL
LIN {X 0,Y 92.868,Z 997.681,A -85,B 0,C 180,E1 3967.793,E2 3967.793} C_VEL
LIN {X 0,Y 110.195,Z 993.803,A -85,B 0,C 180,E1 3956.652,E2 3956.652} C_VEL
LIN {X 0,Y 130.585,Z 988.088,A -85,B 0,C 180,E1 3948.587,E2 3948.587} C_VEL
LIN {X 0,Y 142.248,Z 984.385,A -85,B 0,C 180,E1 3945.158,E2 3945.158} C_VEL
LIN {X 0,Y 119.623,Z 992.322,A -85,B 0,C 180,E1 3938.121,E2 3938.121} C_VEL
LIN {X 0,Y 101.157,Z 997.952,A -85,B 0,C 180,E1 3929.073,E2 3929.073} C_VEL
LIN {X 0,Y 85.27,Z 1002.224,A -85,B 0,C 180,E1 3915.688,E2 3915.688} C_VEL
LIN {X 0,Y 76.211,Z 1004.496,A -85,B 0,C 180,E1 3900.796,E2 3900.796} C_VEL
LIN {X 0,Y 72.302,Z 1005.421,A -85,B 0,C 180,E1 3883.618,E2 3883.618} C_VEL
LIN {X 0,Y 72.108,Z 1005.257,A -85,B 0,C 180,E1 3872.405,E2 3872.405} C_VEL
LIN {X 0,Y 72.098,Z 1004.581,A -85,B 0,C 180,E1 3863.651,E2 3863.651} C_VEL
LIN {X 0,Y 73.288,Z 1002.603,A -85,B 0,C 180,E1 3849.247,E2 3849.247} C_VEL
LIN {X 0,Y 78.476,Z 998.927,A -85,B 0,C 180,E1 3834.146,E2 3834.146} C_VEL
LIN {X 0,Y 84.843,Z 995.37,A -85,B 0,C 180,E1 3824.486,E2 3824.486} C_VEL
LIN {X 0,Y 87.813,Z 993.414,A -85,B 0,C 180,E1 3819.92,E2 3819.92} C_VEL
LIN {X 0,Y 95.012,Z 987.206,A -85,B 0,C 180,E1 3807.955,E2 3807.955} C_VEL
LIN {X 0,Y 98.932,Z 984.949,A -85,B 0,C 180,E1 3805.04,E2 3805.04} C_VEL
LIN {X 0,Y 116.232,Z 975.54,A -85,B 0,C 180,E1 3797.332,E2 3797.332} C_VEL
LIN {X 0,Y 133.83,Z 964.933,A -85,B 0,C 180,E1 3791.907,E2 3791.907} C_VEL
LIN {X 0,Y 151.38,Z 952.801,A -85,B 0,C 180,E1 3787.889,E2 3787.889} C_VEL
LIN {X 0,Y 169.51,Z 938.697,A -85,B 0,C 180,E1 3784.683,E2 3784.683} C_VEL
LIN {X 0,Y 186.095,Z 924.028,A -85,B 0,C 180,E1 3782.337,E2 3782.337} C_VEL
LIN {X 0,Y 202.443,Z 907.561,A -85,B 0,C 180,E1 3780.423,E2 3780.423} C_VEL
LIN {X 0,Y 217.326,Z 890.616,A -85,B 0,C 180,E1 3778.945,E2 3778.945} C_VEL
LIN {X 0,Y 231.617,Z 871.826,A -85,B 0,C 180,E1 3777.716,E2 3777.716} C_VEL
LIN {X 0,Y 244.838,Z 851.985,A -85,B 0,C 180,E1 3776.722,E2 3776.722} C_VEL
LIN {X 0,Y 256.047,Z 832.418,A -85,B 0,C 180,E1 3775.969,E2 3775.969} C_VEL
LIN {X 0,Y 266.816,Z 810.39,A -85,B 0,C 180,E1 3775.32,E2 3775.32} C_VEL
LIN {X 0,Y 276.053,Z 787.829,A -85,B 0,C 180,E1 3774.819,E2 3774.819} C_VEL
LIN {X 0,Y 283.595,Z 764.642,A -85,B 0,C 180,E1 3774.453,E2 3774.453} C_VEL
LIN {X 0,Y 289.882,Z 739.472,A -85,B 0,C 180,E1 3774.122,E2 3774.122} C_VEL
LIN {X 0,Y 294.063,Z 715.625,A -85,B 0,C 180,E1 3773.801,E2 3773.801} C_VEL
LIN {X 0,Y 301.088,Z 663.733,A -85,B 0,C 180,E1 3773.121,E2 3773.121} C_VEL
LIN {X 0,Y 300.419,Z 662.334,A -85,B 0,C 180,E1 3771.579,E2 3771.579} C_VEL
LIN {X 0,Y 299.059,Z 658.328,A -85,B 0,C 180,E1 3764.684,E2 3764.684} C_VEL
LIN {X 0,Y 299.101,Z 658.616,A -85,B 0,C 180,E1 3761.669,E2 3761.669} C_VEL
LIN {X 0,Y 300.879,Z 663.105,A -85,B 0,C 180,E1 3754.615,E2 3754.615} C_VEL
LIN {X 0,Y 300.925,Z 663.506,A -85,B 0,C 180,E1 3754.427,E2 3754.427} C_VEL
LIN {X 0,Y 292.064,Z 726.546,A -85,B 0,C 180,E1 3753.618,E2 3753.618} C_VEL
LIN {X 0,Y 286.845,Z 750.359,A -85,B 0,C 180,E1 3753.291,E2 3753.291} C_VEL
LIN {X 0,Y 279.755,Z 774.69,A -85,B 0,C 180,E1 3752.85,E2 3752.85} C_VEL
LIN {X 0,Y 271.988,Z 795.919,A -85,B 0,C 180,E1 3752.352,E2 3752.352} C_VEL
LIN {X 0,Y 262.292,Z 817.674,A -85,B 0,C 180,E1 3751.696,E2 3751.696} C_VEL
LIN {X 0,Y 251.175,Z 838.867,A -85,B 0,C 180,E1 3750.883,E2 3750.883} C_VEL
LIN {X 0,Y 238.636,Z 859.063,A -85,B 0,C 180,E1 3749.891,E2 3749.891} C_VEL
LIN {X 0,Y 224.247,Z 879.114,A -85,B 0,C 180,E1 3748.616,E2 3748.616} C_VEL
LIN {X 0,Y 209.95,Z 896.517,A -85,B 0,C 180,E1 3747.183,E2 3747.183} C_VEL
LIN {X 0,Y 194.341,Z 913.019,A -85,B 0,C 180,E1 3745.388,E2 3745.388} C_VEL
LIN {X 0,Y 177.517,Z 928.778,A -85,B 0,C 180,E1 3743.095,E2 3743.095} C_VEL
LIN {X 0,Y 160.943,Z 942.34,A -85,B 0,C 180,E1 3740.368,E2 3740.368} C_VEL
LIN {X 0,Y 142.061,Z 955.951,A -85,B 0,C 180,E1 3736.446,E2 3736.446} C_VEL
LIN {X 0,Y 124.729,Z 966.993,A -85,B 0,C 180,E1 3731.691,E2 3731.691} C_VEL
LIN {X 0,Y 107.511,Z 976.581,A -85,B 0,C 180,E1 3725.194,E2 3725.194} C_VEL
LIN {X 0,Y 91.313,Z 984.788,A -85,B 0,C 180,E1 3716.115,E2 3716.115} C_VEL
LIN {X 0,Y 78.541,Z 990.804,A -85,B 0,C 180,E1 3704.637,E2 3704.637} C_VEL
LIN {X 0,Y 68.758,Z 995.702,A -85,B 0,C 180,E1 3688.312,E2 3688.312} C_VEL
LIN {X 0,Y 64.86,Z 998.367,A -85,B 0,C 180,E1 3672.904,E2 3672.904} C_VEL
LIN {X 0,Y 64.119,Z 999.707,A -85,B 0,C 180,E1 3660.845,E2 3660.845} C_VEL
LIN {X 0,Y 64.352,Z 1000.52,A -85,B 0,C 180,E1 3649.236,E2 3649.236} C_VEL
LIN {X 0,Y 66.752,Z 1000.88,A -85,B 0,C 180,E1 3634.493,E2 3634.493} C_VEL
LIN {X 0,Y 74.26,Z 1000.307,A -85,B 0,C 180,E1 3618.042,E2 3618.042} C_VEL
LIN {X 0,Y 89.305,Z 998.026,A -85,B 0,C 180,E1 3602.569,E2 3602.569} C_VEL
LIN {X 0,Y 108.214,Z 994.198,A -85,B 0,C 180,E1 3592.035,E2 3592.035} C_VEL
LIN {X 0,Y 127.503,Z 989.218,A -85,B 0,C 180,E1 3585.239,E2 3585.239} C_VEL
LIN {X 0,Y 103.537,Z 996.312,A -85,B 0,C 180,E1 3576.583,E2 3576.583} C_VEL
LIN {X 0,Y 85.25,Z 1000.933,A -85,B 0,C 180,E1 3565.212,E2 3565.212} C_VEL
LIN {X 0,Y 71.596,Z 1003.798,A -85,B 0,C 180,E1 3548.96,E2 3548.96} C_VEL
LIN {X 0,Y 65.151,Z 1005.029,A -85,B 0,C 180,E1 3530.594,E2 3530.594} C_VEL
LIN {X 0,Y 64.084,Z 1004.997,A -85,B 0,C 180,E1 3515.395,E2 3515.395} C_VEL
LIN {X 0,Y 64.116,Z 1004.431,A -85,B 0,C 180,E1 3506.369,E2 3506.369} C_VEL
LIN {X 0,Y 64.465,Z 1003.215,A -85,B 0,C 180,E1 3494.737,E2 3494.737} C_VEL
LIN {X 0,Y 67.907,Z 1000.553,A -85,B 0,C 180,E1 3479.007,E2 3479.007} C_VEL
LIN {X 0,Y 77.241,Z 995.633,A -85,B 0,C 180,E1 3462.483,E2 3462.483} C_VEL
LIN {X 0,Y 89.688,Z 989.609,A -85,B 0,C 180,E1 3450.849,E2 3450.849} C_VEL
LIN {X 0,Y 98.932,Z 984.949,A -85,B 0,C 180,E1 3445.04,E2 3445.04} C_VEL
LIN {X 0,Y 103.644,Z 982.271,A -85,B 0,C 180,E1 3441.89,E2 3441.89} C_VEL
LIN {X 0,Y 114.968,Z 974.297,A -85,B 0,C 180,E1 3433.412,E2 3433.412} C_VEL
LIN {X 0,Y 119.616,Z 971.348,A -85,B 0,C 180,E1 3431.573,E2 3431.573} C_VEL
LIN {X 0,Y 137.049,Z 960.557,A -85,B 0,C 180,E1 3427.263,E2 3427.263} C_VEL
LIN {X 0,Y 155.299,Z 947.834,A -85,B 0,C 180,E1 3423.863,E2 3423.863} C_VEL
LIN {X 0,Y 171.996,Z 934.523,A -85,B 0,C 180,E1 3421.414,E2 3421.414} C_VEL
LIN {X 0,Y 189.955,Z 918.246,A -85,B 0,C 180,E1 3419.277,E2 3419.277} C_VEL
LIN {X 0,Y 206.105,Z 901.582,A -85,B 0,C 180,E1 3417.688,E2 3417.688} C_VEL
LIN {X 0,Y 221.369,Z 883.383,A -85,B 0,C 180,E1 3416.409,E2 3416.409} C_VEL
LIN {X 0,Y 235.7,Z 863.88,A -85,B 0,C 180,E1 3415.372,E2 3415.372} C_VEL
LIN {X 0,Y 248.035,Z 844.434,A -85,B 0,C 180,E1 3414.589,E2 3414.589} C_VEL
LIN {X 0,Y 259.89,Z 822.561,A -85,B 0,C 180,E1 3413.919,E2 3413.919} C_VEL
LIN {X 0,Y 270.024,Z 800.45,A -85,B 0,C 180,E1 3413.408,E2 3413.408} C_VEL
LIN {X 0,Y 278.126,Z 778.74,A -85,B 0,C 180,E1 3413.037,E2 3413.037} C_VEL
LIN {X 0,Y 285.568,Z 753.779,A -85,B 0,C 180,E1 3412.721,E2 3412.721} C_VEL
LIN {X 0,Y 290.766,Z 730.418,A -85,B 0,C 180,E1 3412.435,E2 3412.435} C_VEL
LIN {X 0,Y 297.634,Z 682.775,A -85,B 0,C 180,E1 3411.846,E2 3411.846} C_VEL
LIN {X 0,Y 299.315,Z 670.324,A -85,B 0,C 180,E1 3411.654,E2 3411.654} C_VEL
LIN {X 0,Y 297.926,Z 666.245,A -85,B 0,C 180,E1 3404.625,E2 3404.625} C_VEL
LIN {X 0,Y 297.955,Z 666.505,A -85,B 0,C 180,E1 3401.815,E2 3401.815} C_VEL
LIN {X 0,Y 299.175,Z 670.373,A -85,B 0,C 180,E1 3395.863,E2 3395.863} C_VEL
LIN {X 0,Y 291.106,Z 727.017,A -85,B 0,C 180,E1 3395.176,E2 3395.176} C_VEL
LIN {X 0,Y 285.848,Z 750.773,A -85,B 0,C 180,E1 3394.877,E2 3394.877} C_VEL
LIN {X 0,Y 278.633,Z 775.293,A -85,B 0,C 180,E1 3394.471,E2 3394.471} C_VEL
LIN {X 0,Y 270.8,Z 796.493,A -85,B 0,C 180,E1 3394.018,E2 3394.018} C_VEL
LIN {X 0,Y 261.015,Z 818.185,A -85,B 0,C 180,E1 3393.422,E2 3393.422} C_VEL
LIN {X 0,Y 249.791,Z 839.333,A -85,B 0,C 180,E1 3392.683,E2 3392.683} C_VEL
LIN {X 0,Y 237.605,Z 858.779,A -85,B 0,C 180,E1 3391.817,E2 3391.817} C_VEL
LIN {X 0,Y 223.18,Z 878.756,A -85,B 0,C 180,E1 3390.673,E2 3390.673} C_VEL
LIN {X 0,Y 208.663,Z 896.27,A -85,B 0,C 180,E1 3389.371,E2 3389.371} C_VEL
LIN {X 0,Y 192.715,Z 912.989,A -85,B 0,C 180,E1 3387.728,E2 3387.728} C_VEL
LIN {X 0,Y 176.539,Z 928.039,A -85,B 0,C 180,E1 3385.763,E2 3385.763} C_VEL
LIN {X 0,Y 159.598,Z 941.72,A -85,B 0,C 180,E1 3383.293,E2 3383.293} C_VEL
LIN {X 0,Y 141.108,Z 954.918,A -85,B 0,C 180,E1 3379.911,E2 3379.911} C_VEL
LIN {X 0,Y 123.999,Z 965.566,A -85,B 0,C 180,E1 3375.841,E2 3375.841} C_VEL
LIN {X 0,Y 105.023,Z 975.933,A -85,B 0,C 180,E1 3369.613,E2 3369.613} C_VEL
LIN {X 0,Y 88.231,Z 984.088,A -85,B 0,C 180,E1 3361.397,E2 3361.397} C_VEL
LIN {X 0,Y 73.579,Z 990.473,A -85,B 0,C 180,E1 3349.838,E2 3349.838} C_VEL
LIN {X 0,Y 62.494,Z 995.448,A -85,B 0,C 180,E1 3333.645,E2 3333.645} C_VEL
LIN {X 0,Y 57.051,Z 998.509,A -85,B 0,C 180,E1 3314.732,E2 3314.732} C_VEL
LIN {X 0,Y 56.121,Z 999.925,A -85,B 0,C 180,E1 3300.815,E2 3300.815} C_VEL
LIN {X 0,Y 56.455,Z 1000.796,A -85,B 0,C 180,E1 3287.666,E2 3287.666} C_VEL
LIN {X 0,Y 59.908,Z 1001.219,A -85,B 0,C 180,E1 3269.74,E2 3269.74} C_VEL
LIN {X 0,Y 69.754,Z 1000.62,A -85,B 0,C 180,E1 3251.579,E2 3251.579} C_VEL
LIN {X 0,Y 87.166,Z 998.287,A -85,B 0,C 180,E1 3236.581,E2 3236.581} C_VEL
LIN {X 0,Y 108.621,Z 994.279,A -85,B 0,C 180,E1 3226.697,E2 3226.697} C_VEL
LIN {X 0,Y 112.682,Z 993.304,A -85,B 0,C 180,E1 3225.326,E2 3225.326} C_VEL
LIN {X 0,Y 89.079,Z 999.09,A -85,B 0,C 180,E1 3215.428,E2 3215.428} C_VEL
LIN {X 0,Y 71.452,Z 1002.643,A -85,B 0,C 180,E1 3201.626,E2 3201.626} C_VEL
LIN {X 0,Y 59.985,Z 1004.397,A -85,B 0,C 180,E1 3182.263,E2 3182.263} C_VEL
LIN {X 0,Y 56.339,Z 1004.717,A -85,B 0,C 180,E1 3164.413,E2 3164.413} C_VEL
LIN {X 0,Y 56.132,Z 1004.387,A -85,B 0,C 180,E1 3152.068,E2 3152.068} C_VEL
LIN {X 0,Y 56.118,Z 1003.758,A -85,B 0,C 180,E1 3141.833,E2 3141.833} C_VEL
LIN {X 0,Y 58.428,Z 1001.378,A -85,B 0,C 180,E1 3122.849,E2 3122.849} C_VEL
LIN {X 0,Y 65.253,Z 997.876,A -85,B 0,C 180,E1 3106.441,E2 3106.441} C_VEL
LIN {X 0,Y 78.395,Z 992.038,A -85,B 0,C 180,E1 3091.333,E2 3091.333} C_VEL
LIN {X 0,Y 93.631,Z 984.985,A -85,B 0,C 180,E1 3081.473,E2 3081.473} C_VEL
LIN {X 0,Y 112.215,Z 975.427,A -85,B 0,C 180,E1 3073.846,E2 3073.846} C_VEL
LIN {X 0,Y 119.616,Z 971.348,A -85,B 0,C 180,E1 3071.573,E2 3071.573} C_VEL
LIN {X 0,Y 125.045,Z 967.822,A -85,B 0,C 180,E1 3069.566,E2 3069.566} C_VEL
LIN {X 0,Y 138.275,Z 958.088,A -85,B 0,C 180,E1 3063.693,E2 3063.693} C_VEL
LIN {X 0,Y 143.169,Z 954.592,A -85,B 0,C 180,E1 3062.516,E2 3062.516} C_VEL
LIN {X 0,Y 160.945,Z 941.713,A -85,B 0,C 180,E1 3059.913,E2 3059.913} C_VEL
LIN {X 0,Y 179.073,Z 926.601,A -85,B 0,C 180,E1 3057.804,E2 3057.804} C_VEL
LIN {X 0,Y 196.025,Z 910.529,A -85,B 0,C 180,E1 3056.197,E2 3056.197} C_VEL
LIN {X 0,Y 211.762,Z 893.3,A -85,B 0,C 180,E1 3054.94,E2 3054.94} C_VEL
LIN {X 0,Y 227.227,Z 873.908,A -85,B 0,C 180,E1 3053.885,E2 3053.885} C_VEL
LIN {X 0,Y 240.768,Z 854.375,A -85,B 0,C 180,E1 3053.082,E2 3053.082} C_VEL
LIN {X 0,Y 252.563,Z 834.426,A -85,B 0,C 180,E1 3052.46,E2 3052.46} C_VEL
LIN {X 0,Y 263.525,Z 812.9,A -85,B 0,C 180,E1 3051.948,E2 3051.948} C_VEL
LIN {X 0,Y 272.653,Z 791.288,A -85,B 0,C 180,E1 3051.564,E2 3051.564} C_VEL
LIN {X 0,Y 280.944,Z 767.149,A -85,B 0,C 180,E1 3051.259,E2 3051.259} C_VEL
LIN {X 0,Y 287.198,Z 743.861,A -85,B 0,C 180,E1 3051.015,E2 3051.015} C_VEL
LIN {X 0,Y 291.659,Z 720.107,A -85,B 0,C 180,E1 3050.742,E2 3050.742} C_VEL
LIN {X 0,Y 297.658,Z 677.505,A -85,B 0,C 180,E1 3050.233,E2 3050.233} C_VEL
LIN {X 0,Y 296.791,Z 674.157,A -85,B 0,C 180,E1 3044.447,E2 3044.447} C_VEL
LIN {X 0,Y 296.811,Z 674.405,A -85,B 0,C 180,E1 3041.945,E2 3041.945} C_VEL
LIN {X 0,Y 297.519,Z 677.53,A -85,B 0,C 180,E1 3037.312,E2 3037.312} C_VEL
LIN {X 0,Y 290.235,Z 727.656,A -85,B 0,C 180,E1 3036.74,E2 3036.74} C_VEL
LIN {X 0,Y 284.902,Z 751.454,A -85,B 0,C 180,E1 3036.468,E2 3036.468} C_VEL
LIN {X 0,Y 277.728,Z 775.576,A -85,B 0,C 180,E1 3036.107,E2 3036.107} C_VEL
LIN {X 0,Y 269.523,Z 797.591,A -85,B 0,C 180,E1 3035.683,E2 3035.683} C_VEL
LIN {X 0,Y 259.481,Z 819.503,A -85,B 0,C 180,E1 3035.137,E2 3035.137} C_VEL
LIN {X 0,Y 247.667,Z 841.301,A -85,B 0,C 180,E1 3034.443,E2 3034.443} C_VEL
LIN {X 0,Y 235.373,Z 860.625,A -85,B 0,C 180,E1 3033.66,E2 3033.66} C_VEL
LIN {X 0,Y 221.153,Z 879.931,A -85,B 0,C 180,E1 3032.654,E2 3032.654} C_VEL
LIN {X 0,Y 206.012,Z 897.917,A -85,B 0,C 180,E1 3031.439,E2 3031.439} C_VEL
LIN {X 0,Y 189.475,Z 914.794,A -85,B 0,C 180,E1 3029.912,E2 3029.912} C_VEL
LIN {X 0,Y 171.128,Z 931.17,A -85,B 0,C 180,E1 3027.889,E2 3027.889} C_VEL
LIN {X 0,Y 153.799,Z 944.687,A -85,B 0,C 180,E1 3025.555,E2 3025.555} C_VEL
LIN {X 0,Y 135.047,Z 957.349,A -85,B 0,C 180,E1 3022.371,E2 3022.371} C_VEL
LIN {X 0,Y 116.614,Z 968.295,A -85,B 0,C 180,E1 3018.219,E2 3018.219} C_VEL
LIN {X 0,Y 98.813,Z 977.36,A -85,B 0,C 180,E1 3012.661,E2 3012.661} C_VEL
LIN {X 0,Y 80.475,Z 985.609,A -85,B 0,C 180,E1 3003.97,E2 3003.97} C_VEL
LIN {X 0,Y 65.773,Z 991.51,A -85,B 0,C 180,E1 2992.311,E2 2992.311} C_VEL
LIN {X 0,Y 53.616,Z 996.4,A -85,B 0,C 180,E1 2973.179,E2 2973.179} C_VEL
LIN {X 0,Y 48.879,Z 998.965,A -85,B 0,C 180,E1 2954.047,E2 2954.047} C_VEL
LIN {X 0,Y 48.109,Z 1000.275,A -85,B 0,C 180,E1 2938.661,E2 2938.661} C_VEL
LIN {X 0,Y 48.924,Z 1001.165,A -85,B 0,C 180,E1 2922.414,E2 2922.414} C_VEL
LIN {X 0,Y 54.539,Z 1001.551,A -85,B 0,C 180,E1 2901.513,E2 2901.513} C_VEL
LIN {X 0,Y 68.08,Z 1000.824,A -85,B 0,C 180,E1 2882.519,E2 2882.519} C_VEL
LIN {X 0,Y 87.784,Z 998.305,A -85,B 0,C 180,E1 2869.502,E2 2869.502} C_VEL
LIN {X 0,Y 97.624,Z 996.696,A -85,B 0,C 180,E1 2865.392,E2 2865.392} C_VEL
LIN {X 0,Y 74.633,Z 1001.176,A -85,B 0,C 180,E1 2853.885,E2 2853.885} C_VEL
LIN {X 0,Y 58.499,Z 1003.59,A -85,B 0,C 180,E1 2837.339,E2 2837.339} C_VEL
LIN {X 0,Y 49.489,Z 1004.399,A -85,B 0,C 180,E1 2813.866,E2 2813.866} C_VEL
LIN {X 0,Y 48.104,Z 1004.137,A -85,B 0,C 180,E1 2795.997,E2 2795.997} C_VEL
LIN {X 0,Y 48.125,Z 1003.64,A -85,B 0,C 180,E1 2785.71,E2 2785.71} C_VEL
LIN {X 0,Y 49.301,Z 1002.008,A -85,B 0,C 180,E1 2767.369,E2 2767.369} C_VEL
LIN {X 0,Y 56.809,Z 998.315,A -85,B 0,C 180,E1 2745.289,E2 2745.289} C_VEL
LIN {X 0,Y 69.207,Z 993.347,A -85,B 0,C 180,E1 2729.954,E2 2729.954} C_VEL
LIN {X 0,Y 85.626,Z 986.39,A -85,B 0,C 180,E1 2719.004,E2 2719.004} C_VEL
LIN {X 0,Y 103.599,Z 977.943,A -85,B 0,C 180,E1 2711.692,E2 2711.692} C_VEL
LIN {X 0,Y 122.276,Z 967.725,A -85,B 0,C 180,E1 2706.572,E2 2706.572} C_VEL
LIN {X 0,Y 141.243,Z 955.929,A -85,B 0,C 180,E1 2702.839,E2 2702.839} C_VEL
LIN {X 0,Y 143.169,Z 954.592,A -85,B 0,C 180,E1 2702.516,E2 2702.516} C_VEL
LIN {X 0,Y 148.809,Z 950.506,A -85,B 0,C 180,E1 2701.207,E2 2701.207} C_VEL
LIN {X 0,Y 162.593,Z 939.036,A -85,B 0,C 180,E1 2697.009,E2 2697.009} C_VEL
LIN {X 0,Y 167.437,Z 934.965,A -85,B 0,C 180,E1 2696.236,E2 2696.236} C_VEL
LIN {X 0,Y 185.259,Z 919.484,A -85,B 0,C 180,E1 2694.614,E2 2694.614} C_VEL
LIN {X 0,Y 201.27,Z 903.499,A -85,B 0,C 180,E1 2693.405,E2 2693.405} C_VEL
LIN {X 0,Y 217.785,Z 884.573,A -85,B 0,C 180,E1 2692.348,E2 2692.348} C_VEL
LIN {X 0,Y 231.973,Z 865.946,A -85,B 0,C 180,E1 2691.572,E2 2691.572} C_VEL
LIN {X 0,Y 244.982,Z 845.953,A -85,B 0,C 180,E1 2690.947,E2 2690.947} C_VEL
LIN {X 0,Y 257.055,Z 824.381,A -85,B 0,C 180,E1 2690.437,E2 2690.437} C_VEL
LIN {X 0,Y 266.928,Z 803.463,A -85,B 0,C 180,E1 2690.067,E2 2690.067} C_VEL
LIN {X 0,Y 275.798,Z 780.678,A -85,B 0,C 180,E1 2689.767,E2 2689.767} C_VEL
LIN {X 0,Y 283.09,Z 757.503,A -85,B 0,C 180,E1 2689.548,E2 2689.548} C_VEL
LIN {X 0,Y 288.512,Z 734.314,A -85,B 0,C 180,E1 2689.326,E2 2689.326} C_VEL
LIN {X 0,Y 293.545,Z 702.91,A -85,B 0,C 180,E1 2688.983,E2 2688.983} C_VEL
LIN {X 0,Y 296.08,Z 684.639,A -85,B 0,C 180,E1 2688.758,E2 2688.758} C_VEL
LIN {X 0,Y 295.658,Z 682.074,A -85,B 0,C 180,E1 2684.303,E2 2684.303} C_VEL
LIN {X 0,Y 295.668,Z 682.304,A -85,B 0,C 180,E1 2682.077,E2 2682.077} C_VEL
LIN {X 0,Y 296.001,Z 684.581,A -85,B 0,C 180,E1 2678.776,E2 2678.776} C_VEL
LIN {X 0,Y 289.506,Z 728.443,A -85,B 0,C 180,E1 2678.309,E2 2678.309} C_VEL
LIN {X 0,Y 284.209,Z 751.89,A -85,B 0,C 180,E1 2678.071,E2 2678.071} C_VEL
LIN {X 0,Y 276.803,Z 776.533,A -85,B 0,C 180,E1 2677.742,E2 2677.742} C_VEL
LIN {X 0,Y 268.612,Z 798.317,A -85,B 0,C 180,E1 2677.369,E2 2677.369} C_VEL
LIN {X 0,Y 258.676,Z 819.779,A -85,B 0,C 180,E1 2676.897,E2 2676.897} C_VEL
LIN {X 0,Y 246.77,Z 841.576,A -85,B 0,C 180,E1 2676.286,E2 2676.286} C_VEL
LIN {X 0,Y 234.373,Z 860.902,A -85,B 0,C 180,E1 2675.598,E2 2675.598} C_VEL
LIN {X 0,Y 220.021,Z 880.208,A -85,B 0,C 180,E1 2674.713,E2 2674.713} C_VEL
LIN {X 0,Y 204.722,Z 898.198,A -85,B 0,C 180,E1 2673.644,E2 2673.644} C_VEL
LIN {X 0,Y 188.478,Z 914.632,A -85,B 0,C 180,E1 2672.344,E2 2672.344} C_VEL
LIN {X 0,Y 170.846,Z 930.321,A -85,B 0,C 180,E1 2670.671,E2 2670.671} C_VEL
LIN {X 0,Y 153.32,Z 943.875,A -85,B 0,C 180,E1 2668.66,E2 2668.66} C_VEL
LIN {X 0,Y 134.035,Z 956.823,A -85,B 0,C 180,E1 2665.873,E2 2665.873} C_VEL
LIN {X 0,Y 115.057,Z 967.899,A -85,B 0,C 180,E1 2662.236,E2 2662.236} C_VEL
LIN {X 0,Y 95.629,Z 977.5,A -85,B 0,C 180,E1 2657.02,E2 2657.02} C_VEL
LIN {X 0,Y 77.108,Z 985.471,A -85,B 0,C 180,E1 2649.421,E2 2649.421} C_VEL
LIN {X 0,Y 61.034,Z 991.441,A -85,B 0,C 180,E1 2638.335,E2 2638.335} C_VEL
LIN {X 0,Y 47.503,Z 996.293,A -85,B 0,C 180,E1 2619.662,E2 2619.662} C_VEL
LIN {X 0,Y 41.108,Z 999.103,A -85,B 0,C 180,E1 2596.651,E2 2596.651} C_VEL
LIN {X 0,Y 40.109,Z 1000.473,A -85,B 0,C 180,E1 2578.39,E2 2578.39} C_VEL
LIN {X 0,Y 41.257,Z 1001.435,A -85,B 0,C 180,E1 2559.063,E2 2559.063} C_VEL
LIN {X 0,Y 49.038,Z 1001.9,A -85,B 0,C 180,E1 2534.166,E2 2534.166} C_VEL
LIN {X 0,Y 65.233,Z 1001.202,A -85,B 0,C 180,E1 2515.311,E2 2515.311} C_VEL
LIN {X 0,Y 82.449,Z 999.358,A -85,B 0,C 180,E1 2505.469,E2 2505.469} C_VEL
LIN {X 0,Y 60.228,Z 1002.581,A -85,B 0,C 180,E1 2491.675,E2 2491.675} C_VEL
LIN {X 0,Y 45.913,Z 1003.941,A -85,B 0,C 180,E1 2470.834,E2 2470.834} C_VEL
LIN {X 0,Y 40.235,Z 1003.917,A -85,B 0,C 180,E1 2442.961,E2 2442.961} C_VEL
LIN {X 0,Y 40.163,Z 1003.385,A -85,B 0,C 180,E1 2428.611,E2 2428.611} C_VEL
LIN {X 0,Y 40.666,Z 1002.199,A -85,B 0,C 180,E1 2411.399,E2 2411.399} C_VEL
LIN {X 0,Y 46.823,Z 999.329,A -85,B 0,C 180,E1 2386.942,E2 2386.942} C_VEL
LIN {X 0,Y 60.06,Z 994.475,A -85,B 0,C 180,E1 2368.133,E2 2368.133} C_VEL
LIN {X 0,Y 77.093,Z 988.069,A -85,B 0,C 180,E1 2356.388,E2 2356.388} C_VEL
LIN {X 0,Y 96.096,Z 979.709,A -85,B 0,C 180,E1 2348.833,E2 2348.833} C_VEL
LIN {X 0,Y 116.193,Z 969.502,A -85,B 0,C 180,E1 2343.683,E2 2343.683} C_VEL
LIN {X 0,Y 134.119,Z 958.91,A -85,B 0,C 180,E1 2340.426,E2 2340.426} C_VEL
LIN {X 0,Y 154.071,Z 945.299,A -85,B 0,C 180,E1 2337.699,E2 2337.699} C_VEL
LIN {X 0,Y 167.437,Z 934.965,A -85,B 0,C 180,E1 2336.236,E2 2336.236} C_VEL
LIN {X 0,Y 172.982,Z 930.275,A -85,B 0,C 180,E1 2335.357,E2 2335.357} C_VEL
LIN {X 0,Y 185.783,Z 917.896,A -85,B 0,C 180,E1 2332.349,E2 2332.349} C_VEL
LIN {X 0,Y 191.139,Z 912.641,A -85,B 0,C 180,E1 2331.683,E2 2331.683} C_VEL
LIN {X 0,Y 207.656,Z 895.269,A -85,B 0,C 180,E1 2330.718,E2 2330.718} C_VEL
LIN {X 0,Y 222.98,Z 876.865,A -85,B 0,C 180,E1 2329.958,E2 2329.958} C_VEL
LIN {X 0,Y 237.012,Z 857.193,A -85,B 0,C 180,E1 2329.354,E2 2329.354} C_VEL
LIN {X 0,Y 250.143,Z 835.803,A -85,B 0,C 180,E1 2328.861,E2 2328.861} C_VEL
LIN {X 0,Y 261.172,Z 814.749,A -85,B 0,C 180,E1 2328.499,E2 2328.499} C_VEL
LIN {X 0,Y 270.624,Z 792.917,A -85,B 0,C 180,E1 2328.223,E2 2328.223} C_VEL
LIN {X 0,Y 278.922,Z 769.657,A -85,B 0,C 180,E1 2328.018,E2 2328.018} C_VEL
LIN {X 0,Y 285.165,Z 747.228,A -85,B 0,C 180,E1 2327.852,E2 2327.852} C_VEL
LIN {X 0,Y 290.141,Z 722.742,A -85,B 0,C 180,E1 2327.623,E2 2327.623} C_VEL
LIN {X 0,Y 294.683,Z 691.734,A -85,B 0,C 180,E1 2327.289,E2 2327.289} C_VEL
LIN {X 0,Y 294.527,Z 689.994,A -85,B 0,C 180,E1 2324.241,E2 2324.241} C_VEL
LIN {X 0,Y 294.527,Z 690.203,A -85,B 0,C 180,E1 2322.209,E2 2322.209} C_VEL
LIN {X 0,Y 294.612,Z 691.686,A -85,B 0,C 180,E1 2320.254,E2 2320.254} C_VEL
LIN {X 0,Y 288.859,Z 729.46,A -85,B 0,C 180,E1 2319.884,E2 2319.884} C_VEL
LIN {X 0,Y 283.548,Z 752.697,A -85,B 0,C 180,E1 2319.676,E2 2319.676} C_VEL
LIN {X 0,Y 276.349,Z 776.471,A -85,B 0,C 180,E1 2319.399,E2 2319.399} C_VEL
LIN {X 0,Y 268.108,Z 798.297,A -85,B 0,C 180,E1 2319.077,E2 2319.077} C_VEL
LIN {X 0,Y 258.112,Z 819.846,A -85,B 0,C 180,E1 2318.669,E2 2318.669} C_VEL
LIN {X 0,Y 246.627,Z 840.9,A -85,B 0,C 180,E1 2318.165,E2 2318.165} C_VEL
LIN {X 0,Y 234.077,Z 860.437,A -85,B 0,C 180,E1 2317.573,E2 2317.573} C_VEL
LIN {X 0,Y 219.175,Z 880.433,A -85,B 0,C 180,E1 2316.791,E2 2316.791} C_VEL
LIN {X 0,Y 203.738,Z 898.458,A -85,B 0,C 180,E1 2315.874,E2 2315.874} C_VEL
LIN {X 0,Y 187.822,Z 914.445,A -85,B 0,C 180,E1 2314.798,E2 2314.798} C_VEL
LIN {X 0,Y 169.975,Z 930.212,A -85,B 0,C 180,E1 2313.372,E2 2313.372} C_VEL
LIN {X 0,Y 152.191,Z 943.804,A -85,B 0,C 180,E1 2311.66,E2 2311.66} C_VEL
LIN {X 0,Y 132.55,Z 956.817,A -85,B 0,C 180,E1 2309.283,E2 2309.283} C_VEL
LIN {X 0,Y 113.11,Z 967.934,A -85,B 0,C 180,E1 2306.168,E2 2306.168} C_VEL
LIN {X 0,Y 93.032,Z 977.599,A -85,B 0,C 180,E1 2301.652,E2 2301.652} C_VEL
LIN {X 0,Y 73.226,Z 985.755,A -85,B 0,C 180,E1 2294.759,E2 2294.759} C_VEL
LIN {X 0,Y 55.432,Z 991.894,A -85,B 0,C 180,E1 2283.964,E2 2283.964} C_VEL
LIN {X 0,Y 39.726,Z 996.867,A -85,B 0,C 180,E1 2263.053,E2 2263.053} C_VEL
LIN {X 0,Y 33.096,Z 999.422,A -85,B 0,C 180,E1 2237.745,E2 2237.745} C_VEL
LIN {X 0,Y 32.108,Z 1000.694,A -85,B 0,C 180,E1 2217.234,E2 2217.234} C_VEL
LIN {X 0,Y 33.821,Z 1001.705,A -85,B 0,C 180,E1 2194.054,E2 2194.054} C_VEL
LIN {X 0,Y 44.511,Z 1002.251,A -85,B 0,C 180,E1 2165.159,E2 2165.159} C_VEL
LIN {X 0,Y 63.877,Z 1001.572,A -85,B 0,C 180,E1 2147.344,E2 2147.344} C_VEL
LIN {X 0,Y 67.061,Z 1001.305,A -85,B 0,C 180,E1 2145.489,E2 2145.489} C_VEL
LIN {X 0,Y 45.89,Z 1003.308,A -85,B 0,C 180,E1 2128.242,E2 2128.242} C_VEL
LIN {X 0,Y 34.429,Z 1003.691,A -85,B 0,C 180,E1 2101.566,E2 2101.566} C_VEL
LIN {X 0,Y 32.131,Z 1003.182,A -85,B 0,C 180,E1 2075.333,E2 2075.333} C_VEL
LIN {X 0,Y 32.134,Z 1002.709,A -85,B 0,C 180,E1 2062.898,E2 2062.898} C_VEL
LIN {X 0,Y 35.535,Z 1000.564,A -85,B 0,C 180,E1 2033.834,E2 2033.834} C_VEL
LIN {X 0,Y 45.931,Z 997.117,A -85,B 0,C 180,E1 2011.492,E2 2011.492} C_VEL
LIN {X 0,Y 63.425,Z 991.4,A -85,B 0,C 180,E1 1996.018,E2 1996.018} C_VEL
LIN {X 0,Y 81.83,Z 984.391,A -85,B 0,C 180,E1 1987.722,E2 1987.722} C_VEL
LIN {X 0,Y 103.016,Z 974.864,A -85,B 0,C 180,E1 1981.967,E2 1981.967} C_VEL
LIN {X 0,Y 121.993,Z 964.851,A -85,B 0,C 180,E1 1978.525,E2 1978.525} C_VEL
LIN {X 0,Y 141.376,Z 952.855,A -85,B 0,C 180,E1 1975.943,E2 1975.943} C_VEL
LIN {X 0,Y 159.803,Z 939.823,A -85,B 0,C 180,E1 1974.06,E2 1974.06} C_VEL
LIN {X 0,Y 178.032,Z 924.766,A -85,B 0,C 180,E1 1972.577,E2 1972.577} C_VEL
LIN {X 0,Y 191.139,Z 912.641,A -85,B 0,C 180,E1 1971.683,E2 1971.683} C_VEL
LIN {X 0,Y 196.434,Z 907.359,A -85,B 0,C 180,E1 1971.061,E2 1971.061} C_VEL
LIN {X 0,Y 208.611,Z 893.609,A -85,B 0,C 180,E1 1968.725,E2 1968.725} C_VEL
LIN {X 0,Y 213.423,Z 887.774,A -85,B 0,C 180,E1 1968.248,E2 1968.248} C_VEL
LIN {X 0,Y 227.644,Z 869.671,A -85,B 0,C 180,E1 1967.718,E2 1967.718} C_VEL
LIN {X 0,Y 241.889,Z 848.735,A -85,B 0,C 180,E1 1967.258,E2 1967.258} C_VEL
LIN {X 0,Y 253.496,Z 828.859,A -85,B 0,C 180,E1 1966.931,E2 1966.931} C_VEL
LIN {X 0,Y 264.042,Z 807.405,A -85,B 0,C 180,E1 1966.67,E2 1966.67} C_VEL
LIN {X 0,Y 273.052,Z 785.669,A -85,B 0,C 180,E1 1966.472,E2 1966.472} C_VEL
LIN {X 0,Y 280.617,Z 762.747,A -85,B 0,C 180,E1 1966.336,E2 1966.336} C_VEL
LIN {X 0,Y 286.958,Z 737.733,A -85,B 0,C 180,E1 1966.173,E2 1966.173} C_VEL
LIN {X 0,Y 291.269,Z 713.794,A -85,B 0,C 180,E1 1965.959,E2 1965.959} C_VEL
LIN {X 0,Y 293.387,Z 698.789,A -85,B 0,C 180,E1 1965.795,E2 1965.795} C_VEL
LIN {X 0,Y 293.398,Z 697.916,A -85,B 0,C 180,E1 1963.976,E2 1963.976} C_VEL
LIN {X 0,Y 293.386,Z 698.246,A -85,B 0,C 180,E1 1962.138,E2 1962.138} C_VEL
LIN {X 0,Y 293.37,Z 698.681,A -85,B 0,C 180,E1 1961.745,E2 1961.745} C_VEL
LIN {X 0,Y 288.198,Z 731.36,A -85,B 0,C 180,E1 1961.458,E2 1961.458} C_VEL
LIN {X 0,Y 282.889,Z 754.227,A -85,B 0,C 180,E1 1961.281,E2 1961.281} C_VEL
LIN {X 0,Y 275.623,Z 777.777,A -85,B 0,C 180,E1 1961.045,E2 1961.045} C_VEL
LIN {X 0,Y 267.036,Z 800.17,A -85,B 0,C 180,E1 1960.761,E2 1960.761} C_VEL
LIN {X 0,Y 257.294,Z 820.877,A -85,B 0,C 180,E1 1960.43,E2 1960.43} C_VEL
LIN {X 0,Y 245.241,Z 842.601,A -85,B 0,C 180,E1 1959.988,E2 1959.988} C_VEL
LIN {X 0,Y 232.679,Z 861.917,A -85,B 0,C 180,E1 1959.494,E2 1959.494} C_VEL
LIN {X 0,Y 218.115,Z 881.176,A -85,B 0,C 180,E1 1958.861,E2 1958.861} C_VEL
LIN {X 0,Y 202.56,Z 899.133,A -85,B 0,C 180,E1 1958.098,E2 1958.098} C_VEL
LIN {X 0,Y 186.509,Z 915.087,A -85,B 0,C 180,E1 1957.206,E2 1957.206} C_VEL
LIN {X 0,Y 168.481,Z 930.817,A -85,B 0,C 180,E1 1956.026,E2 1956.026} C_VEL
LIN {X 0,Y 150.484,Z 944.401,A -85,B 0,C 180,E1 1954.611,E2 1954.611} C_VEL
LIN {X 0,Y 130.548,Z 957.377,A -85,B 0,C 180,E1 1952.649,E2 1952.649} C_VEL
LIN {X 0,Y 110.725,Z 968.482,A -85,B 0,C 180,E1 1950.068,E2 1950.068} C_VEL
LIN {X 0,Y 90.1,Z 978.105,A -85,B 0,C 180,E1 1946.301,E2 1946.301} C_VEL
LIN {X 0,Y 69.863,Z 986.084,A -85,B 0,C 180,E1 1940.572,E2 1940.572} C_VEL
LIN {X 0,Y 51.368,Z 992.062,A -85,B 0,C 180,E1 1931.396,E2 1931.396} C_VEL
LIN {X 0,Y 34.192,Z 996.911,A -85,B 0,C 180,E1 1912.295,E2 1912.295} C_VEL
LIN {X 0,Y 25.246,Z 999.666,A -85,B 0,C 180,E1 1880.825,E2 1880.825} C_VEL
LIN {X 0,Y 24.112,Z 1000.888,A -85,B 0,C 180,E1 1856.044,E2 1856.044} C_VEL
LIN {X 0,Y 27.326,Z 1002.021,A -85,B 0,C 180,E1 1823.698,E2 1823.698} C_VEL
LIN {X 0,Y 42.418,Z 1002.602,A -85,B 0,C 180,E1 1793.236,E2 1793.236} C_VEL
LIN {X 0,Y 51.549,Z 1002.509,A -85,B 0,C 180,E1 1785.601,E2 1785.601} C_VEL
LIN {X 0,Y 31.728,Z 1003.352,A -85,B 0,C 180,E1 1762.057,E2 1762.057} C_VEL
LIN {X 0,Y 24.385,Z 1002.951,A -85,B 0,C 180,E1 1726.743,E2 1726.743} C_VEL
LIN {X 0,Y 24.163,Z 1002.52,A -85,B 0,C 180,E1 1707.691,E2 1707.691} C_VEL
LIN {X 0,Y 26.877,Z 1000.779,A -85,B 0,C 180,E1 1673.543,E2 1673.543} C_VEL
LIN {X 0,Y 39.608,Z 997.11,A -85,B 0,C 180,E1 1644.758,E2 1644.758} C_VEL
LIN {X 0,Y 57.9,Z 991.787,A -85,B 0,C 180,E1 1630.316,E2 1630.316} C_VEL
LIN {X 0,Y 78.043,Z 984.567,A -85,B 0,C 180,E1 1622.646,E2 1622.646} C_VEL
LIN {X 0,Y 99.02,Z 975.598,A -85,B 0,C 180,E1 1617.948,E2 1617.948} C_VEL
LIN {X 0,Y 118.394,Z 965.698,A -85,B 0,C 180,E1 1615.054,E2 1615.054} C_VEL
LIN {X 0,Y 139.042,Z 953.314,A -85,B 0,C 180,E1 1612.813,E2 1612.813} C_VEL
LIN {X 0,Y 157.903,Z 940.199,A -85,B 0,C 180,E1 1611.258,E2 1611.258} C_VEL
LIN {X 0,Y 175.56,Z 925.917,A -85,B 0,C 180,E1 1610.095,E2 1610.095} C_VEL
LIN {X 0,Y 192.882,Z 910.012,A -85,B 0,C 180,E1 1609.16,E2 1609.16} C_VEL
LIN {X 0,Y 209.196,Z 892.607,A -85,B 0,C 180,E1 1608.419,E2 1608.419} C_VEL
LIN {X 0,Y 213.423,Z 887.774,A -85,B 0,C 180,E1 1608.248,E2 1608.248} C_VEL
LIN {X 0,Y 218.14,Z 881.902,A -85,B 0,C 180,E1 1607.794,E2 1607.794} C_VEL
LIN {X 0,Y 229.917,Z 865.999,A -85,B 0,C 180,E1 1605.816,E2 1605.816} C_VEL
LIN {X 0,Y 233.658,Z 860.552,A -85,B 0,C 180,E1 1605.537,E2 1605.537} C_VEL
LIN {X 0,Y 246.372,Z 840.819,A -85,B 0,C 180,E1 1605.252,E2 1605.252} C_VEL
LIN {X 0,Y 257.668,Z 820.082,A -85,B 0,C 180,E1 1605.036,E2 1605.036} C_VEL
LIN {X 0,Y 267.744,Z 798.346,A -85,B 0,C 180,E1 1604.871,E2 1604.871} C_VEL
LIN {X 0,Y 275.876,Z 776.885,A -85,B 0,C 180,E1 1604.761,E2 1604.761} C_VEL
LIN {X 0,Y 283.37,Z 752.024,A -85,B 0,C 180,E1 1604.66,E2 1604.66} C_VEL
LIN {X 0,Y 288.724,Z 728.402,A -85,B 0,C 180,E1 1604.506,E2 1604.506} C_VEL
LIN {X 0,Y 292.266,Z 705.835,A -85,B 0,C 180,E1 1604.269,E2 1604.269} C_VEL
LIN {X 0,Y 292.226,Z 705.982,A -85,B 0,C 180,E1 1603.248,E2 1603.248} C_VEL
LIN {X 0,Y 287.479,Z 734.196,A -85,B 0,C 180,E1 1603.032,E2 1603.032} C_VEL
LIN {X 0,Y 281.796,Z 757.88,A -85,B 0,C 180,E1 1602.879,E2 1602.879} C_VEL
LIN {X 0,Y 274.364,Z 780.964,A -85,B 0,C 180,E1 1602.683,E2 1602.683} C_VEL
LIN {X 0,Y 264.99,Z 804.363,A -85,B 0,C 180,E1 1602.43,E2 1602.43} C_VEL
LIN {X 0,Y 254.703,Z 825.662,A -85,B 0,C 180,E1 1602.141,E2 1602.141} C_VEL
LIN {X 0,Y 243.094,Z 845.772,A -85,B 0,C 180,E1 1601.8,E2 1601.8} C_VEL
LIN {X 0,Y 229.968,Z 865.491,A -85,B 0,C 180,E1 1601.383,E2 1601.383} C_VEL
LIN {X 0,Y 215.828,Z 883.693,A -85,B 0,C 180,E1 1600.893,E2 1600.893} C_VEL
LIN {X 0,Y 198.662,Z 902.856,A -85,B 0,C 180,E1 1600.22,E2 1600.22} C_VEL
LIN {X 0,Y 181.495,Z 919.483,A -85,B 0,C 180,E1 1599.448,E2 1599.448} C_VEL
LIN {X 0,Y 163.315,Z 934.556,A -85,B 0,C 180,E1 1598.496,E2 1598.496} C_VEL
LIN {X 0,Y 144.137,Z 948.403,A -85,B 0,C 180,E1 1597.277,E2 1597.277} C_VEL
LIN {X 0,Y 124.977,Z 960.255,A -85,B 0,C 180,E1 1595.755,E2 1595.755} C_VEL
LIN {X 0,Y 103.844,Z 971.363,A -85,B 0,C 180,E1 1593.529,E2 1593.529} C_VEL
LIN {X 0,Y 82.803,Z 980.668,A -85,B 0,C 180,E1 1590.35,E2 1590.35} C_VEL
LIN {X 0,Y 61.95,Z 988.097,A -85,B 0,C 180,E1 1585.353,E2 1585.353} C_VEL
LIN {X 0,Y 41.638,Z 994.052,A -85,B 0,C 180,E1 1576.033,E2 1576.033} C_VEL
LIN {X 0,Y 24.929,Z 997.982,A -85,B 0,C 180,E1 1556.111,E2 1556.111} C_VEL
LIN {X 0,Y 16.854,Z 1000.159,A -85,B 0,C 180,E1 1519.658,E2 1519.658} C_VEL
LIN {X 0,Y 16.278,Z 1001.214,A -85,B 0,C 180,E1 1487.371,E2 1487.371} C_VEL
LIN {X 0,Y 24.199,Z 1002.449,A -85,B 0,C 180,E1 1442.376,E2 1442.376} C_VEL
LIN {X 0,Y 35.51,Z 1002.976,A -85,B 0,C 180,E1 1425.597,E2 1425.597} C_VEL
LIN {X 0,Y 18.67,Z 1002.741,A -85,B 0,C 180,E1 1390.094,E2 1390.094} C_VEL
LIN {X 0,Y 16.197,Z 1002.1,A -85,B 0,C 180,E1 1350.093,E2 1350.093} C_VEL
LIN {X 0,Y 19.689,Z 1000.479,A -85,B 0,C 180,E1 1304.797,E2 1304.797} C_VEL
LIN {X 0,Y 35.1,Z 996.814,A -85,B 0,C 180,E1 1274.593,E2 1274.593} C_VEL
LIN {X 0,Y 55.026,Z 991.492,A -85,B 0,C 180,E1 1262.723,E2 1262.723} C_VEL
LIN {X 0,Y 76.074,Z 984.271,A -85,B 0,C 180,E1 1256.865,E2 1256.865} C_VEL
LIN {X 0,Y 97.615,Z 975.302,A -85,B 0,C 180,E1 1253.342,E2 1253.342} C_VEL
LIN {X 0,Y 117.381,Z 965.383,A -85,B 0,C 180,E1 1251.179,E2 1251.179} C_VEL
LIN {X 0,Y 138.261,Z 953.02,A -85,B 0,C 180,E1 1249.508,E2 1249.508} C_VEL
LIN {X 0,Y 157.184,Z 939.98,A -85,B 0,C 180,E1 1248.351,E2 1248.351} C_VEL
LIN {X 0,Y 175.165,Z 925.534,A -85,B 0,C 180,E1 1247.471,E2 1247.471} C_VEL
LIN {X 0,Y 192.383,Z 909.807,A -85,B 0,C 180,E1 1246.78,E2 1246.78} C_VEL
LIN {X 0,Y 208.424,Z 892.791,A -85,B 0,C 180,E1 1246.234,E2 1246.234} C_VEL
LIN {X 0,Y 224.84,Z 872.747,A -85,B 0,C 180,E1 1245.764,E2 1245.764} C_VEL
LIN {X 0,Y 233.658,Z 860.552,A -85,B 0,C 180,E1 1245.537,E2 1245.537} C_VEL
LIN {X 0,Y 233.489,Z 860.748,A -85,B 0,C 180,E1 1245.298,E2 1245.298} C_VEL
LIN {X 0,Y 231.582,Z 863.437,A -85,B 0,C 180,E1 1244.79,E2 1244.79} C_VEL
LIN {X 0,Y 226.119,Z 870.77,A -85,B 0,C 180,E1 1244.033,E2 1244.033} C_VEL
LIN {X 0,Y 217.34,Z 881.917,A -85,B 0,C 180,E1 1243.173,E2 1243.173} C_VEL
LIN {X 0,Y 212.772,Z 887.402,A -85,B 0,C 180,E1 1242.936,E2 1242.936} C_VEL
LIN {X 0,Y 196.566,Z 904.946,A -85,B 0,C 180,E1 1242.473,E2 1242.473} C_VEL
LIN {X 0,Y 178.796,Z 921.729,A -85,B 0,C 180,E1 1241.895,E2 1241.895} C_VEL
LIN {X 0,Y 161.518,Z 935.838,A -85,B 0,C 180,E1 1241.25,E2 1241.25} C_VEL
LIN {X 0,Y 141.178,Z 950.184,A -85,B 0,C 180,E1 1240.343,E2 1240.343} C_VEL
LIN {X 0,Y 120.824,Z 962.495,A -85,B 0,C 180,E1 1239.206,E2 1239.206} C_VEL
LIN {X 0,Y 100.201,Z 972.876,A -85,B 0,C 180,E1 1237.715,E2 1237.715} C_VEL
LIN {X 0,Y 78.02,Z 982.221,A -85,B 0,C 180,E1 1235.44,E2 1235.44} C_VEL
LIN {X 0,Y 57.629,Z 989.145,A -85,B 0,C 180,E1 1232.174,E2 1232.174} C_VEL
LIN {X 0,Y 34.732,Z 995.218,A -85,B 0,C 180,E1 1224.841,E2 1224.841} C_VEL
LIN {X 0,Y 17.654,Z 998.698,A -85,B 0,C 180,E1 1208.426,E2 1208.426} C_VEL
LIN {X 0,Y 8.33,Z 1000.688,A -85,B 0,C 180,E1 1153.873,E2 1153.873} C_VEL
LIN {X 0,Y 10.377,Z 1001.683,A -85,B 0,C 180,E1 1094.978,E2 1094.978} C_VEL
LIN {X 0,Y 19.03,Z 1002.566,A -85,B 0,C 180,E1 1065.975,E2 1065.975} C_VEL
LIN {X 0,Y 8.173,Z 1001.662,A -85,B 0,C 180,E1 997.212,E2 997.212} C_VEL
LIN {X 0,Y 9.98,Z 1000.786,A -85,B 0,C 180,E1 945.679,E2 945.679} C_VEL
LIN {X 0,Y 27.082,Z 997.595,A -85,B 0,C 180,E1 905.23,E2 905.23} C_VEL
LIN {X 0,Y 47.08,Z 992.823,A -85,B 0,C 180,E1 895.995,E2 895.995} C_VEL
LIN {X 0,Y 68.855,Z 986.166,A -85,B 0,C 180,E1 891.648,E2 891.648} C_VEL
LIN {X 0,Y 89.523,Z 978.168,A -85,B 0,C 180,E1 889.271,E2 889.271} C_VEL
LIN {X 0,Y 111.571,Z 967.823,A -85,B 0,C 180,E1 887.578,E2 887.578} C_VEL
LIN {X 0,Y 131.602,Z 956.637,A -85,B 0,C 180,E1 886.473,E2 886.473} C_VEL
LIN {X 0,Y 150.645,Z 944.115,A -85,B 0,C 180,E1 885.654,E2 885.654} C_VEL
LIN {X 0,Y 169.729,Z 929.703,A -85,B 0,C 180,E1 884.999,E2 884.999} C_VEL
LIN {X 0,Y 187.209,Z 914.264,A -85,B 0,C 180,E1 884.511,E2 884.511} C_VEL
LIN {X 0,Y 204.773,Z 896.491,A -85,B 0,C 180,E1 884.1,E2 884.1} C_VEL
LIN {X 0,Y 219.65,Z 879.123,A -85,B 0,C 180,E1 883.807,E2 883.807} C_VEL
LIN {X 0,Y 233.994,Z 859.748,A -85,B 0,C 180,E1 883.565,E2 883.565} C_VEL
LIN {X 0,Y 235.915,Z 856.934,A -85,B 0,C 180,E1 883.526,E2 883.526} C_VEL
LIN {X 0,Y 221.929,Z 876.235,A -85,B 0,C 180,E1 883.181,E2 883.181} C_VEL
LIN {X 0,Y 212.772,Z 887.402,A -85,B 0,C 180,E1 882.936,E2 882.936} C_VEL
LIN {X 0,Y 212.312,Z 888.681,A -85,B 0,C 180,E1 882.922,E2 882.922} C_VEL
LIN {X 0,Y 212.312,Z 902.944,A -85,B 0,C 180,E1 882.922,E2 882.922} C_VEL
LIN {X 0,Y 188.705,Z 926.391,A -85,B 0,C 180,E1 882.977,E2 882.977} C_VEL
LIN {X 0,Y 162.859,Z 947.48,A -85,B 0,C 180,E1 883.054,E2 883.054} C_VEL
LIN {X 0,Y 135.309,Z 965.751,A -85,B 0,C 180,E1 883.17,E2 883.17} C_VEL
LIN {X 0,Y 133.52,Z 965.964,A -85,B 0,C 180,E1 883.179,E2 883.179} C_VEL
LIN {X 0,Y 128.616,Z 964.181,A -85,B 0,C 180,E1 883.205,E2 883.205} C_VEL
LIN {X 0,Y 127.3,Z 962.301,A -85,B 0,C 180,E1 883.213,E2 883.213} C_VEL
LIN {X 0,Y 127.3,Z 962.301,A -85,B 0,C 180,E1 883.213,E2 883.213} C_VEL
LIN {X 0,Y 124.306,Z 960.569,A -85,B 0,C 180,E1 883.124,E2 883.124} C_VEL
LIN {X 0,Y 102.482,Z 971.873,A -85,B 0,C 180,E1 882.393,E2 882.393} C_VEL
LIN {X 0,Y 81.153,Z 981.083,A -85,B 0,C 180,E1 881.501,E2 881.501} C_VEL
LIN {X 0,Y 59.361,Z 988.586,A -85,B 0,C 180,E1 880.31,E2 880.31} C_VEL
LIN {X 0,Y 37.562,Z 994.562,A -85,B 0,C 180,E1 878.582,E2 878.582} C_VEL
LIN {X 0,Y 17.021,Z 998.601,A -85,B 0,C 180,E1 875.708,E2 875.708} C_VEL
LIN {X 0,Y 3.429,Z 1000.595,A -85,B 0,C 180,E1 870.109,E2 870.109} C_VEL
LIN {X 0,Y 0.321,Z 1001.049,A -85,B 0,C 180,E1 1049.255,E2 1049.255} C_VEL
LIN {X 0,Y 14.195,Z 999.188,A -85,B 0,C 180,E1 889.817,E2 889.817} C_VEL
LIN {X 0,Y 32.771,Z 995.744,A -85,B 0,C 180,E1 887.29,E2 887.29} C_VEL
LIN {X 0,Y 56.273,Z 989.703,A -85,B 0,C 180,E1 885.593,E2 885.593} C_VEL
LIN {X 0,Y 76.711,Z 982.855,A -85,B 0,C 180,E1 884.611,E2 884.611} C_VEL
LIN {X 0,Y 98.875,Z 973.628,A -85,B 0,C 180,E1 883.817,E2 883.817} C_VEL
LIN {X 0,Y 118.993,Z 963.579,A -85,B 0,C 180,E1 883.265,E2 883.265} C_VEL
LIN {X 0,Y 124.306,Z 960.569,A -85,B 0,C 180,E1 883.124,E2 883.124} C_VEL
LIN {X 0,Y 125.02,Z 962.531,A -85,B 0,C 180,E1 882.076,E2 882.076} C_VEL
LIN {X 0,Y 125.02,Z 1028,A -85,B 0,C 180,E1 882.076,E2 882.076} C_VEL
LIN {X 0,Y 125.02,Z 1028,A -85,B 0,C 180,E1 882.076,E2 882.076}

QRS_NEXT_CUT()

QRS_NEXT()
QRS_HOME()

END
